stInitSubModulesException.etDiag											:= GD.ET_Diag.UnexpectedProgramBehavior;
stInitSubModulesException.udiDiagExt										:= ET_DiagExt.InitSubModulesException;
stInitSubModulesException.sDiagExt											:= FC_EtDiagExtToString(stInitSubModulesException.udiDiagExt);
stInitSubModulesException.sMsg												:= '';	(* Replaced on usage *)
stInitSubModulesException.udiModuleId										:= iq_stStandardModuleItf.i_udiModuleId;
stInitSubModulesException.sModuleName										:= iq_stStandardModuleItf.i_sModuleName;
stInitSubModulesException.stReaction.axReaction[TPL.ET_Reaction.AsyncStop]	:= TRUE;
stInitSubModulesException.etSource											:= TPL.ET_ExceptionSource.NodeModule;
stInitSubModulesException.timDelayTime										:= T#0MS;
stInitSubModulesException.wHmiAttributes									:= 0;
stInitSubModulesException.xAutoQuit											:= FALSE;

stIsDriveVirtualException.etDiag											:= GD.ET_Diag.InputParameterInvalid;
stIsDriveVirtualException.udiDiagExt										:= ET_DiagExt.ifMulticarrierSegmentsInvalid ;
stIsDriveVirtualException.sDiagExt											:= FC_EtDiagExtToString(stIsDriveVirtualException.udiDiagExt);
stIsDriveVirtualException.sMsg												:= '';	(* Replaced on usage *)
stIsDriveVirtualException.udiModuleId										:= iq_stStandardModuleItf.i_udiModuleId;
stIsDriveVirtualException.sModuleName										:= iq_stStandardModuleItf.i_sModuleName;
stIsDriveVirtualException.stReaction.axReaction[TPL.ET_Reaction.AsyncStop]	:= TRUE;
stIsDriveVirtualException.etSource											:= TPL.ET_ExceptionSource.NodeModule;
stIsDriveVirtualException.timDelayTime										:= T#0MS;
stIsDriveVirtualException.wHmiAttributes									:= 0;
stIsDriveVirtualException.xAutoQuit											:= FALSE;

(*------------------------------------------------------------------------------------------*)
(* Init User Exceptions *)

	// TPL.ET_Reaction.AsyncStop
	// TPL.ET_Reaction.SyncStopEL
	// TPL.ET_Reaction.SyncStopEH
	// TPL.ET_Reaction.StopEndOfCycle
	// TPL.ET_Reaction.MainsContactorOff

(*------------------------------------------------------------------------------------------*)
stUserException1.etDiag													:= GD.ET_Diag.ExecutionAborted;
stUserException1.udiDiagExt												:= ET_DiagExtUser.Exception1FromEquipmentModule;
stUserException1.sDiagExt												:= FC_EtDiagExtUserToString(stUserException1.udiDiagExt);
stUserException1.sMsg													:= 'User Exception 1';
stUserException1.udiModuleId											:= iq_stStandardModuleItf.i_udiModuleId;
stUserException1.sModuleName											:= iq_stStandardModuleItf.i_sModuleName;
stUserException1.stReaction.axReaction[TPL.Gc_udiUserReactionOffset+2]	:= TRUE;
stUserException1.etSource												:= TPL.ET_ExceptionSource.User;
stUserException1.timDelayTime											:= T#0MS;
stUserException1.wHmiAttributes											:= 0;
stUserException1.xAutoQuit												:= FALSE;

stUserException2.etDiag													:= GD.ET_Diag.ExecutionAborted;
stUserException2.udiDiagExt												:= ET_DiagExtUser.Exception2FromEquipmentModule;
stUserException2.sDiagExt												:= FC_EtDiagExtUserToString(stUserException2.udiDiagExt);
stUserException2.sMsg													:= 'User Exception 2';
stUserException2.udiModuleId											:= iq_stStandardModuleItf.i_udiModuleId;
stUserException2.sModuleName											:= iq_stStandardModuleItf.i_sModuleName;
stUserException2.stReaction.axReaction[TPL.Gc_udiUserReactionOffset+2]	:= TRUE;
stUserException2.etSource												:= TPL.ET_ExceptionSource.User;
stUserException2.timDelayTime											:= T#0MS;
stUserException2.wHmiAttributes											:= 0;
stUserException2.xAutoQuit												:= FALSE;

(* End of system generated code, could be modified for your application *)
END_ACTION

ACTION Init_Reactions:
(* System generated code, only to be changed by experienced programmers *)
IF c_udiNumberOfSubModules < 1 THEN
	RETURN;
END_IF

(* Change of default reactions only on demand *)
(* Compare SR MainMachine Action Init_Reactions *)

xInitReactionsException := FALSE;

(*****************************************************************************************************************************************************)
(* Init ReactionTranslationMode *)

TPL.FC_InitReactionTranslationMode(	i_udiNumberOfSubModules			:= c_udiNumberOfSubModules,
									i_petReactionTranslationMode	:= ADR(aetReactionTranslationMode),
									q_etDiag						=> etDiag,
									q_etDiagExt						=> etDiagExtTPL);
							
IF etDiag <> GD.ET_Diag.Ok AND NOT xInitReactionsException THEN
	xInitReactionsException := TRUE;
	
	stInitReactionsException.sMsg := PDL.FC_MultiConcat(i_sString1 := 'InitReactionTranslationMode - ', 
														i_sString2 := GD.FC_EtDiagToString(i_etDiag := etDiag), 
														i_sString3 := ' - ', 
														i_sString4 := TPL.FC_EtDiagExtToString(i_etDiagExt := etDiagExtTPL));
END_IF	

(*****************************************************************************************************************************************************)
(* Init ReactionTranslationTable *)	

TPL.FC_InitReactionTranslationTable(i_udiNumberOfSubModules			:= c_udiNumberOfSubModules,
									i_pstReactionTranslationTable	:= ADR(aastReactionTranslationTable),
									q_etDiag						=> etDiag,
									q_etDiagExt						=> etDiagExtTPL);
									
IF etDiag <> GD.ET_Diag.Ok AND NOT xInitReactionsException THEN
	xInitReactionsException := TRUE;
	
	stInitReactionsException.sMsg := PDL.FC_MultiConcat(i_sString1 := 'InitReactionTranslationTable - ', 
														i_sString2 := GD.FC_EtDiagToString(i_etDiag := etDiag), 
														i_sString3 := ' - ', 
														i_sString4 := TPL.FC_EtDiagExtToString(i_etDiagExt := etDiagExtTPL));
END_IF		

(*****************************************************************************************************************************************************)
(* Init ReactionTranslationJobs *)	
					
TPL.FC_InitReactionTranslationJobs( i_udiNumberOfSubModules			:= c_udiNumberOfSubModules,
									i_pstReactionTranslationJobs	:= ADR(astReactionTranslationJobs),
									q_etDiag						=> etDiag,
									q_etDiagExt						=> etDiagExtTPL);
						
IF etDiag <> GD.ET_Diag.Ok AND NOT xInitReactionsException THEN
	xInitReactionsException := TRUE;
	
	stInitReactionsException.sMsg := PDL.FC_MultiConcat(i_sString1 := 'InitReactionTranslationJobs - ', 
														i_sString2 := GD.FC_EtDiagToString(i_etDiag := etDiag), 
														i_sString3 := ' - ', 
														i_sString4 := TPL.FC_EtDiagExtToString(i_etDiagExt := etDiagExtTPL));
END_IF		

(*****************************************************************************************************************************************************)
(* Set exception if any exception occurred *)
fbExceptionHandler.SetException(i_xExceptionActive	:= xInitReactionsException, 
								iq_stException		:= stInitReactionsException, 
								iq_stExceptionList	:= iq_stExceptionList);
		
xInitSuccessful := xInitSuccessful AND NOT xInitReactionsException;

etDiag := GD.ET_Diag.Ok;
(* End of system generated code, only to be changed by experienced programmers *)
END_ACTION

ACTION ModuleFaults:
(* System generated code, could be modified for your application *)
(* User Exception *)
fbExceptionHandler.SetException(	i_xExceptionActive	:= xModuleUserException1,
									iq_stException		:= stUserException1,
									iq_stExceptionList	:= iq_stExceptionList,
									q_etDiag			=> ,
									q_etDiagExt			=> ,
									q_sMsg				=> );

fbExceptionHandler.SetException(	i_xExceptionActive	:= xModuleUserException2,
									iq_stException		:= stUserException2,
									iq_stExceptionList	:= iq_stExceptionList,
									q_etDiag			=> ,
									q_etDiagExt			=> ,
									q_sMsg				=> );

(* end of System generated code, could be modified for your application *)
END_ACTION

METHOD RegisterLoggerPoint
VAR_INPUT
	i_ifParent	: APL.IF_LoggerPoint;
	i_sName		: STRING[80];
END_VAR
VAR_OUTPUT
	q_etDiag	: GD.ET_Diag := GD.ET_Diag.Ok;
	q_etDiagExt	: ET_DiagExt := ET_DiagExt.Ok;
END_VAR
fbLoggerPoint.RegisterLoggerPoint(	i_ifParent	:= i_ifParent,
									i_sName		:= i_sName,
									i_sType		:= 'Node Module',
									i_sSource	:= 'Program',
									q_etDiag	=> ,
									q_etDiagExt	=> );
END_METHOD

ACTION InitModule_Action:
(* This step is used for initialisations after being enabled *)

(* System generated code, could be modified for your application *)
Init_Exceptions();
(* End of system generated code, could be modified for your application *)

(* System generated code, do not change without consulting 'Schneider Electric Automation GmbH' - otherwise you risk instability!!!*)
xInitSuccessful := TRUE;
xIsDriveVirtualException := FALSE;

iq_stStandardModuleItf.q_xActive		:= TRUE;
iq_stStandardModuleItf.q_xReady			:= FALSE;
iq_stStandardModuleItf.q_etDiag			:= GD.ET_Diag.Ok;
iq_stStandardModuleItf.q_udiDiagExt		:= ET_DiagExt.Initializing;
iq_stStandardModuleItf.q_sDiagExt		:= FC_EtDiagExtToString(ET_DiagExt.Initializing);
iq_stStandardModuleItf.q_sMsg			:= '';
			
Init_SubModules();
Init_CmdTables();
Init_Reactions();
UpdateStructs();
(* End of system generated code, do not change without consulting 'Schneider Electric Automation GmbH' - otherwise you risk instability!!!*)

(* System generated code, could be modified for your application *)
fbModuleController.RegisterLoggerPoint(	i_ifParent	:= fbLoggerPoint,
										i_sName		:= 'ModuleController',
										q_etDiag	=> ,
										q_etDiagExt	=> );
fbExceptionHandler.RegisterLoggerPoint(	i_ifParent	:= fbLoggerPoint,
										i_sName		:= 'ExceptionHandler',
										q_etDiag	=> ,
										q_etDiagExt	=> );
										
Init_Master();
(* End of system generated code, could be modified for your application *)

(* Application specific code *)
(* ToDo: Add your application specific code here *)
;
(* End of application specific code *)
END_ACTION

ACTION Input_Action:
(* System generated code, do not change without consulting 'Schneider Electric Automation GmbH' - otherwise you risk instability!!!*)
UpdateStructs();
(* End of system generated code, do not change without consulting 'Schneider Electric Automation GmbH' - otherwise you risk instability!!!*)
END_ACTION

ACTION Logger_Action:
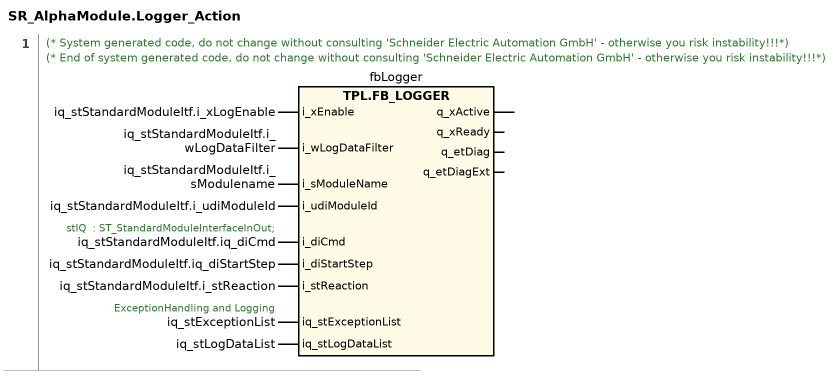
// NETWORK 1
// 					(* System generated code, do not change without consulting 'Schneider Electric Automation GmbH' - otherwise you risk instability!!!*)
// (* End of system generated code, do not change without consulting 'Schneider Electric Automation GmbH' - otherwise you risk instability!!!*)
//
//   fbLogger: Logging related variables
//   iq_stStandardModuleItf.iq_diCmd: stIQ : ST_StandardModuleInterfaceInOut;
//   iq_stExceptionList: ExceptionHandling and Logging
fbLogger(
    i_xEnable := iq_stStandardModuleItf.i_xLogEnable,
    i_wLogDataFilter := iq_stStandardModuleItf.i_wLogDataFilter,
    i_sModuleName := iq_stStandardModuleItf.i_sModulename,
    i_udiModuleId := iq_stStandardModuleItf.i_udiModuleId,
    i_diCmd := iq_stStandardModuleItf.iq_diCmd,
    i_diStartStep := iq_stStandardModuleItf.iq_diStartStep,
    i_stReaction := iq_stStandardModuleItf.i_stReaction,
    iq_stExceptionList := iq_stExceptionList,
    iq_stLogDataList := iq_stLogDataList); // TPL.FB_LOGGER
END_ACTION

ACTION Logic_active:
Check_RTB();
END_ACTION

ACTION Output_Active:
(* System generated code, only to be changed by experienced programmers *)
IF iq_stStandardModuleItf.q_udiSubModuleInException <> 0 THEN
	iq_stStandardModuleItf.q_etDiag		:= GD.ET_Diag.Ok;
	iq_stStandardModuleItf.q_udiDiagExt	:= ET_DiagExt.SubModuleInException;
	iq_stStandardModuleItf.q_sDiagExt		:= FC_EtDiagExtToString(ET_DiagExt.SubModuleInException);
	iq_stStandardModuleItf.q_sMsg			:= '';
ELSE
	IF etDiagModuleController = GD.ET_Diag.Ok THEN
		iq_stStandardModuleItf.q_etDiag	:= etDiagModuleController;
		iq_stStandardModuleItf.q_sMsg		:= sMsgModuleController;
		
		CASE etDiagExtModuleController OF
			TPL.ET_DiagExt.DeactivatingSubModules : 
				iq_stStandardModuleItf.q_udiDiagExt	:= ET_DiagExt.DeactivatingSubModules;
				iq_stStandardModuleItf.q_sDiagExt		:= FC_EtDiagExtToString(ET_DiagExt.DeactivatingSubModules);
			TPL.ET_DiagExt.Disabled : 
				iq_stStandardModuleItf.q_udiDiagExt	:= ET_DiagExt.Disabled;
				iq_stStandardModuleItf.q_sDiagExt		:= FC_EtDiagExtToString(ET_DiagExt.Disabled);
			TPL.ET_DiagExt.ExecuteStep : 
				iq_stStandardModuleItf.q_udiDiagExt	:= ET_DiagExt.ExecuteStep;
				iq_stStandardModuleItf.q_sDiagExt		:= FC_EtDiagExtToString(ET_DiagExt.ExecuteStep);
			TPL.ET_DiagExt.Initializing : 
				iq_stStandardModuleItf.q_udiDiagExt	:= ET_DiagExt.Initializing;
				iq_stStandardModuleItf.q_sDiagExt		:= FC_EtDiagExtToString(ET_DiagExt.Initializing);
			TPL.ET_DiagExt.WaitAtNegativeStep : 
				iq_stStandardModuleItf.q_udiDiagExt	:= ET_DiagExt.WaitAtNegativeStep;
				iq_stStandardModuleItf.q_sDiagExt		:= FC_EtDiagExtToString(ET_DiagExt.WaitAtNegativeStep);
			TPL.ET_DiagExt.WaitCmdsDone : 
				iq_stStandardModuleItf.q_udiDiagExt	:= ET_DiagExt.WaitCmdsDone;
				iq_stStandardModuleItf.q_sDiagExt		:= FC_EtDiagExtToString(ET_DiagExt.WaitCmdsDone);
			TPL.ET_DiagExt.WaitForCmd : 
				iq_stStandardModuleItf.q_udiDiagExt	:= ET_DiagExt.WaitForCmd;
				iq_stStandardModuleItf.q_sDiagExt		:= FC_EtDiagExtToString(ET_DiagExt.WaitForCmd);
			ELSE
				iq_stStandardModuleItf.q_etDiag		:= GD. ET_Diag.UnexpectedProgramBehavior;
				iq_stStandardModuleItf.q_udiDiagExt	:= ET_DiagExt.UnknownStateModuleController;
				iq_stStandardModuleItf.q_sDiagExt		:= FC_EtDiagExtToString(ET_DiagExt.UnknownStateModuleController);
		END_CASE
	ELSE
		iq_stStandardModuleItf.q_etDiag		:= GD.ET_Diag.DiagActive;
		iq_stStandardModuleItf.q_udiDiagExt	:= ET_DiagExt.ModuleControllerException;
		iq_stStandardModuleItf.q_sDiagExt		:= FC_EtDiagExtToString(ET_DiagExt.ModuleControllerException);
		iq_stStandardModuleItf.q_sMsg			:= PDL.FC_MultiConcat(	i_sString1 := GD.FC_EtDiagToString(i_etDiag := etDiagModuleController), 
																			i_sString2 := ' - ',
																			i_sString3 := TPL.FC_EtDiagExtToString(etDiagExtModuleController), 
																			i_sString4 := '');
	END_IF
END_IF

(* End of system generated code, only to be changed by experienced programmers *)
END_ACTION

ACTION Start_Action:
(* This step is active until the machine is being enabled *)

(* System generated code, do not change without consulting 'Schneider Electric Automation GmbH' - otherwise you risk instability!!! *)
iq_stStandardModuleItf.q_xActive			:= FALSE;
iq_stStandardModuleItf.q_xReady				:= FALSE;

iq_stStandardModuleItf.q_etDiag				:= GD.ET_Diag.Ok;
iq_stStandardModuleItf.q_udiDiagExt			:= ET_DiagExt.Disabled;
iq_stStandardModuleItf.q_sDiagExt			:= FC_EtDiagExtToString(iq_stStandardModuleItf.q_udiDiagExt);
iq_stStandardModuleItf.q_sMsg				:= '';

iq_stStandardModuleItf.q_dwModuleType		:= TPL.ET_ModuleType.NodeModule;
iq_stStandardModuleItf.q_sModuleTypeName	:= 'NodeModule';
iq_stStandardModuleItf.q_udiModuleVersion	:= 1;	
(* End of system generated code, do not change without consulting 'Schneider Electric Automation GmbH' - otherwise you risk instability!!! *)

(* System generated code, to be changed by experienced programmers *)
IF iq_stStandardModuleItf.iq_diCmd <> 0 AND NOT iq_stStandardModuleItf.i_xEnable THEN
	iq_stStandardModuleItf.iq_diCmd := 0;
END_IF
(* End of system generated code, to be changed by experienced programmers *)

(* Application specific code *)
(* ToDo: Add your application specific code here *)
;
(* End of application specific code *)
END_ACTION

ACTION SubModules_Action:
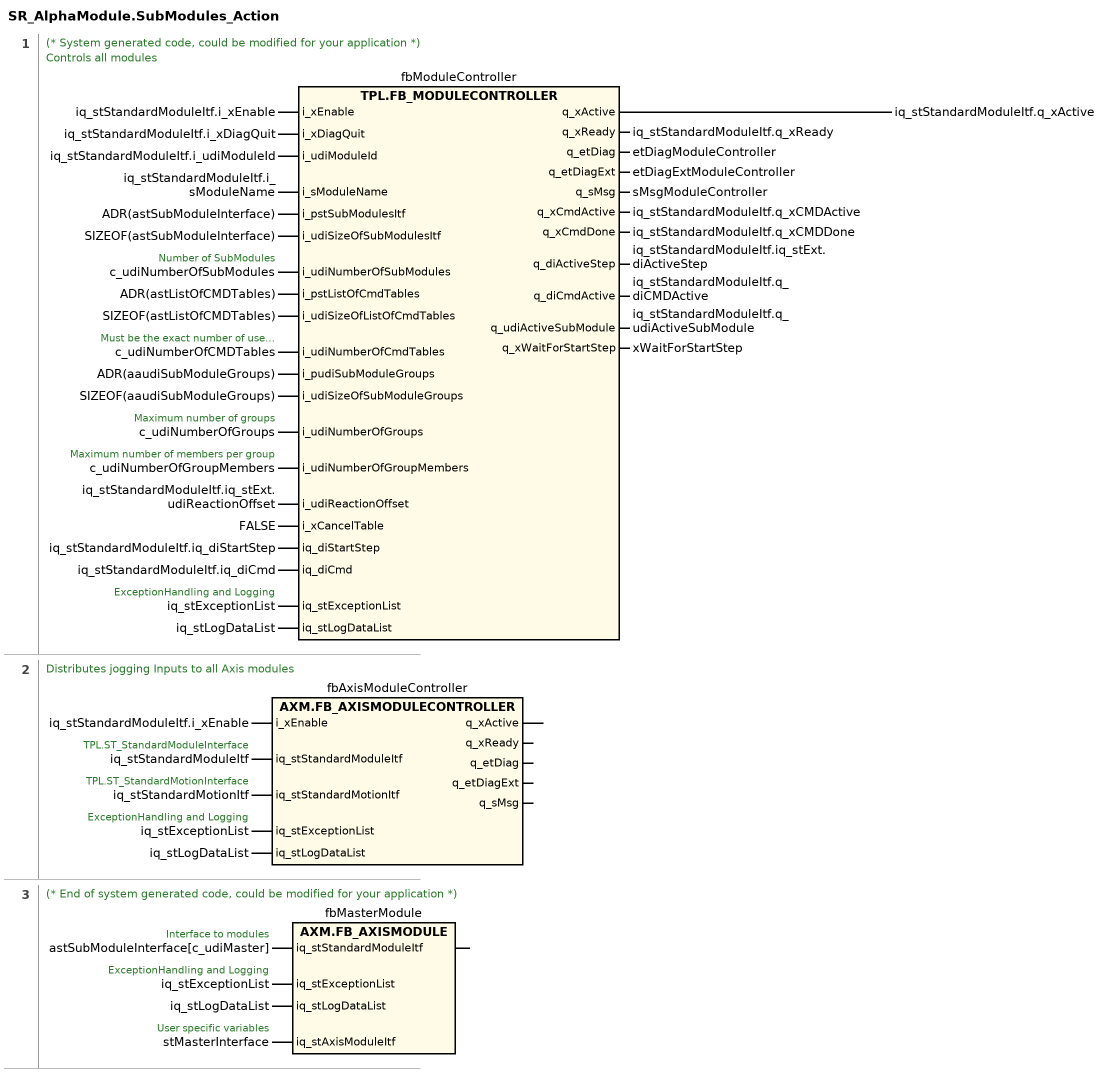
// NETWORK 1
// 					(* System generated code, could be modified for your application *)
// Controls all modules
//
//   fbModuleController: Modules related variables
//   c_udiNumberOfSubModules: Number of SubModules
//   c_udiNumberOfCMDTables: Must be the exact number of used CmdTables!
//   c_udiNumberOfGroups: Maximum number of groups
//   c_udiNumberOfGroupMembers: Maximum number of members per group
//   iq_stExceptionList: ExceptionHandling and Logging
fbModuleController(
    i_xEnable := iq_stStandardModuleItf.i_xEnable,
    i_xDiagQuit := iq_stStandardModuleItf.i_xDiagQuit,
    i_udiModuleId := iq_stStandardModuleItf.i_udiModuleId,
    i_sModuleName := iq_stStandardModuleItf.i_sModuleName,
    i_pstSubModulesItf := ADR(astSubModuleInterface),
    i_udiSizeOfSubModulesItf := SIZEOF(astSubModuleInterface),
    i_udiNumberOfSubModules := c_udiNumberOfSubModules,
    i_pstListOfCmdTables := ADR(astListOfCMDTables),
    i_udiSizeOfListOfCmdTables := SIZEOF(astListOfCMDTables),
    i_udiNumberOfCmdTables := c_udiNumberOfCMDTables,
    i_pudiSubModuleGroups := ADR(aaudiSubModuleGroups),
    i_udiSizeOfSubModuleGroups := SIZEOF(aaudiSubModuleGroups),
    i_udiNumberOfGroups := c_udiNumberOfGroups,
    i_udiNumberOfGroupMembers := c_udiNumberOfGroupMembers,
    i_udiReactionOffset := iq_stStandardModuleItf.iq_stExt.udiReactionOffset,
    i_xCancelTable := FALSE,
    iq_diStartStep := iq_stStandardModuleItf.iq_diStartStep,
    iq_diCmd := iq_stStandardModuleItf.iq_diCmd,
    iq_stExceptionList := iq_stExceptionList,
    iq_stLogDataList := iq_stLogDataList,
    q_xReady => iq_stStandardModuleItf.q_xReady,
    q_etDiag => etDiagModuleController,
    q_etDiagExt => etDiagExtModuleController,
    q_sMsg => sMsgModuleController,
    q_xCmdActive => iq_stStandardModuleItf.q_xCMDActive,
    q_xCmdDone => iq_stStandardModuleItf.q_xCMDDone,
    q_diActiveStep => iq_stStandardModuleItf.iq_stExt.diActiveStep,
    q_diCmdActive => iq_stStandardModuleItf.q_diCMDActive,
    q_udiActiveSubModule => iq_stStandardModuleItf.q_udiActiveSubModule,
    q_xWaitForStartStep => xWaitForStartStep); // TPL.FB_MODULECONTROLLER
iq_stStandardModuleItf.q_xActive := fbModuleController.q_xActive;

// NETWORK 2
// Distributes jogging Inputs to all Axis modules
//   iq_stStandardModuleItf: TPL.ST_StandardModuleInterface
//   iq_stStandardMotionItf: TPL.ST_StandardMotionInterface
//   iq_stExceptionList: ExceptionHandling and Logging
fbAxisModuleController(
    i_xEnable := iq_stStandardModuleItf.i_xEnable,
    iq_stStandardModuleItf := iq_stStandardModuleItf,
    iq_stStandardMotionItf := iq_stStandardMotionItf,
    iq_stExceptionList := iq_stExceptionList,
    iq_stLogDataList := iq_stLogDataList); // AXM.FB_AXISMODULECONTROLLER

// NETWORK 3
// (* End of system generated code, could be modified for your application *)
//   astSubModuleInterface[c_udiMaster]: Interface to modules
//   iq_stExceptionList: ExceptionHandling and Logging
//   stMasterInterface: User specific variables
fbMasterModule(
    iq_stStandardModuleItf := astSubModuleInterface[c_udiMaster],
    iq_stExceptionList := iq_stExceptionList,
    iq_stLogDataList := iq_stLogDataList,
    iq_stAxisModuleItf := stMasterInterface); // AXM.FB_AXISMODULE
END_ACTION

ACTION UpdateStructs:
(* System generated code, do not change without consulting 'Schneider Electric Automation GmbH' - otherwise you risk instability!!! *)
fbDetectOnlineChange(	i_xEnable	:= TRUE, 
						i_xDetect	:= TRUE, 
						q_xActive	=> xDetectOnlineChangeActive, 
						q_xReady	=> xDetectOnlineChangeReady, 
						q_etDiag	=> etDetectOnlineChangeDiag, 
						q_etDiagExt	=> etDetectOnlineChangeDiagExt, 
						q_sMsg		=> sDetectOnlineChangeMsg, 
						q_xChange	=> );
						
IF(NOT fbDetectOnlineChange.q_xChange) THEN
	RETURN;
END_IF

iq_stStandardModuleItf.iq_stExt.udiNumberOfSubModules 		:= c_udiNumberOfSubModules;
iq_stStandardModuleItf.iq_stExt.dwSubModulesItf		 		:= ADR(astSubModuleInterface);
iq_stStandardModuleItf.iq_stExt.pdwSubModulesAddItf		 	:= ADR(adwSubModuleAddInterfaces);
iq_stStandardModuleItf.iq_stExt.pstListOfCmdTables			:= ADR(astListOfCmdTables);
iq_stStandardModuleItf.iq_stExt.udiNumberOfCmdTables		:= c_udiNumberOfCmdTables;
(* End of system generated code, do not change without consulting 'Schneider Electric Automation GmbH' - otherwise you risk instability!!! *)

(* System generated code, could be modified for your application *)
xUpdateStructsException := FALSE;

//-------------------------------------------------------------------------------------------------------------------
//-- Update CmdTable - Prepare 
	//
	TPL.FC_UpdateCmdTableListElement(	i_pstListofCmdTables	:= ADR(astListOfCmdTables),
										i_udiNumberOfCmdTables	:= c_udiNumberOfCmdTables,
										i_diCmd					:= ET_Cmd.Prepare,
										i_pstCmdTable			:= ADR(astPrepareTable),
										q_etDiag				=> etDiag,
										q_etDiagExt				=> etDiagExtTPL);
										
	IF etDiag <> GD.ET_Diag.Ok AND NOT xUpdateStructsException THEN
		xUpdateStructsException := TRUE;
		
		stUpdateStructsException.sMsg := PDL.FC_MultiConcat(i_sString1 := 'Update CmdTable: Prepare - ', 
															i_sString2 := GD.FC_EtDiagToString(i_etDiag := etDiag), 
															i_sString3 := ' - ', 
															i_sString4 := TPL.FC_EtDiagExtToString(i_etDiagExt := etDiagExtTPL));
	END_IF										

//-------------------------------------------------------------------------------------------------------------------
//-- Update CmdTable - Auto 
	//
	TPL.FC_UpdateCmdTableListElement(	i_pstListofCmdTables	:= ADR(astListOfCmdTables),
										i_udiNumberOfCmdTables	:= c_udiNumberOfCmdTables,
										i_diCmd					:= ET_Cmd.Auto,
										i_pstCmdTable			:= ADR(astAutoTable),
										q_etDiag				=> etDiag,
										q_etDiagExt				=> etDiagExtTPL);
										
	IF etDiag <> GD.ET_Diag.Ok AND NOT xUpdateStructsException THEN
		xUpdateStructsException := TRUE;
		
		stUpdateStructsException.sMsg := PDL.FC_MultiConcat(i_sString1 := 'Update CmdTable: Auto - ', 
															i_sString2 := GD.FC_EtDiagToString(i_etDiag := etDiag), 
															i_sString3 := ' - ', 
															i_sString4 := TPL.FC_EtDiagExtToString(i_etDiagExt := etDiagExtTPL));
	END_IF		

//-------------------------------------------------------------------------------------------------------------------
//-- Update CmdTable - Manual 
	//
	TPL.FC_UpdateCmdTableListElement(	i_pstListofCMDTables	:= ADR(astListofCMDTables),
										i_udiNumberOfCMDTables	:= c_udiNumberOfCMDTables,
										i_diCMD					:= ET_Cmd.Manual,
										i_pstCMDTable			:= ADR(astManualTable),
										q_etDiag				=> etDiag,
										q_etDiagExt				=> etDiagExtTPL);
										
	IF etDiag <> GD.ET_Diag.Ok AND NOT xUpdateStructsException THEN
		xUpdateStructsException := TRUE;
		
		stUpdateStructsException.sMsg := PDL.FC_MultiConcat(i_sString1 := 'Update CmdTable: Manual - ', 
															i_sString2 := GD.FC_EtDiagToString(i_etDiag := etDiag), 
															i_sString3 := ' - ', 
															i_sString4 := TPL.FC_EtDiagExtToString(i_etDiagExt := etDiagExtTPL));
	END_IF		

//-------------------------------------------------------------------------------------------------------------------
//-- Update CmdTable - Stop 
	//
	TPL.FC_UpdateCmdTableListElement(	i_pstListofCMDTables	:= ADR(astListofCMDTables),
										i_udiNumberOfCMDTables	:= c_udiNumberOfCMDTables,
										i_diCMD					:= ET_Cmd.Stop,
										i_pstCMDTable			:= ADR(astStopTable),
										q_etDiag				=> etDiag,
										q_etDiagExt				=> etDiagExtTPL);
										
	IF etDiag <> GD.ET_Diag.Ok AND NOT xUpdateStructsException THEN
		xUpdateStructsException := TRUE;
		
		stUpdateStructsException.sMsg := PDL.FC_MultiConcat(i_sString1 := 'Update CmdTable: Stop - ', 
															i_sString2 := GD.FC_EtDiagToString(i_etDiag := etDiag), 
															i_sString3 := ' - ', 
															i_sString4 := TPL.FC_EtDiagExtToString(i_etDiagExt := etDiagExtTPL));
	END_IF		

//-------------------------------------------------------------------------------------------------------------------
//-- Update CmdTable - Start 
	//
	TPL.FC_UpdateCmdTableListElement(	i_pstListofCMDTables	:= ADR(astListofCMDTables),
										i_udiNumberOfCmdTables	:= c_udiNumberOfCMDTables,
										i_diCMD					:= ET_Cmd.Start,
										i_pstCMDTable			:= ADR(astStartTable),
										q_etDiag				=> etDiag,
										q_etDiagExt				=> etDiagExtTPL);
										
	IF etDiag <> GD.ET_Diag.Ok AND NOT xUpdateStructsException THEN
		xUpdateStructsException := TRUE;
		
		stUpdateStructsException.sMsg := PDL.FC_MultiConcat(i_sString1 := 'Update CmdTable: Start - ', 
															i_sString2 := GD.FC_EtDiagToString(i_etDiag := etDiag), 
															i_sString3 := ' - ', 
															i_sString4 := TPL.FC_EtDiagExtToString(i_etDiagExt := etDiagExtTPL));
	END_IF		

//-------------------------------------------------------------------------------------------------------------------
//-- Update CmdTable - Abort 
	//
	TPL.FC_UpdateCmdTableListElement(	i_pstListofCMDTables	:= ADR(astListofCMDTables),
										i_udiNumberOfCmdTables	:= c_udiNumberOfCmdTables,
										i_diCMD					:= ET_Cmd.Abort,
										i_pstCMDTable			:= ADR(astAbortTable),
										q_etDiag				=> etDiag,
										q_etDiagExt				=> etDiagExtTPL);
										
	IF etDiag <> GD.ET_Diag.Ok AND NOT xUpdateStructsException THEN
		xUpdateStructsException := TRUE;
		
		stUpdateStructsException.sMsg := PDL.FC_MultiConcat(i_sString1 := 'Update CmdTable: Abort - ', 
															i_sString2 := GD.FC_EtDiagToString(i_etDiag := etDiag), 
															i_sString3 := ' - ', 
															i_sString4 := TPL.FC_EtDiagExtToString(i_etDiagExt := etDiagExtTPL));
	END_IF		

//-------------------------------------------------------------------------------------------------------------------
//-- Update CmdTable - Hold 
	//
	TPL.FC_UpdateCmdTableListElement(	i_pstListofCMDTables	:= ADR(astListofCMDTables),
										i_udiNumberOfCmdTables	:= c_udiNumberOfCmdTables,
										i_diCMD					:= ET_Cmd.Hold,
										i_pstCMDTable			:= ADR(astHoldTable),
										q_etDiag				=> etDiag,
										q_etDiagExt				=> etDiagExtTPL);
										
	IF etDiag <> GD.ET_Diag.Ok AND NOT xUpdateStructsException THEN
		xUpdateStructsException := TRUE;
		
		stUpdateStructsException.sMsg := PDL.FC_MultiConcat(i_sString1 := 'Update CmdTable: Hold - ', 
															i_sString2 := GD.FC_EtDiagToString(i_etDiag := etDiag), 
															i_sString3 := ' - ', 
															i_sString4 := TPL.FC_EtDiagExtToString(i_etDiagExt := etDiagExtTPL));
	END_IF		

//-------------------------------------------------------------------------------------------------------------------
//-- Update CmdTable - BrakeRelease 
	//
	TPL.FC_UpdateCmdTableListElement(	i_pstListofCMDTables	:= ADR(astListofCMDTables),
										i_udiNumberOfCMDTables	:= c_udiNumberOfCMDTables,
										i_diCMD					:= ET_Cmd.BrakeRelease,
										i_pstCMDTable			:= ADR(astBrakeReleaseTable),
										q_etDiag				=> etDiag,
										q_etDiagExt				=> etDiagExtTPL);
										
	IF etDiag <> GD.ET_Diag.Ok AND NOT xUpdateStructsException THEN
		xUpdateStructsException := TRUE;
		
		stUpdateStructsException.sMsg := PDL.FC_MultiConcat(i_sString1 := 'Update CmdTable: BrakeRelease - ', 
															i_sString2 := GD.FC_EtDiagToString(i_etDiag := etDiag), 
															i_sString3 := ' - ', 
															i_sString4 := TPL.FC_EtDiagExtToString(i_etDiagExt := etDiagExtTPL));
	END_IF		
									
//-------------------------------------------------------------------------------------------------------------------
//-- Update AddInterface - Master 
	//

	AXM.FC_UpdateAddInterfaceStruct(	i_pdwSubModuleAddInterfaces	:= ADR(adwSubModuleAddInterfaces),
										i_udiSubModuleConstant		:= c_udiMaster,
										iq_stAxisModuleItf			:= stMasterInterface,
										q_etDiag					=> etDiag,
										q_etDiagExt					=> etDiagExtAXM);
										
	IF etDiag <> GD.ET_Diag.Ok AND NOT xUpdateStructsException THEN
		xUpdateStructsException := TRUE;
		
		stUpdateStructsException.sMsg := PDL.FC_MultiConcat(i_sString1 := 'Update AddInterface: Master - ', 
															i_sString2 := GD.FC_EtDiagToString(i_etDiag := etDiag), 
															i_sString3 := ' - ', 
															i_sString4 := AXM.FC_EtDiagExtToString(i_etDiagExt := etDiagExtAXM));
	END_IF		

//-------------------------------------------------------------------------------------------------------------------
//-- Update ILS Data 
	//
	// stMasterInterface.stEndless.pstIlsData	:= ADR(G_stIlsData);
	// stMasterInterface.stMultiCam.pstIlsData	:= ADR(G_stIlsData);

//-------------------------------------------------------------------------------------------------------------------
//-- Set exception if any exception occurred *)

fbExceptionHandler.SetException(i_xExceptionActive	:= xUpdateStructsException, 
								iq_stException		:= stUpdateStructsException, 
								iq_stExceptionList	:= iq_stExceptionList);
					
xInitSuccessful := xInitSuccessful AND NOT xUpdateStructsException;

etDiag := GD.ET_Diag.Ok;
(* End of system generated code, could be modified for your application *)
END_ACTION

END_PROGRAM

// LMC_PacDrive/Application/TemplateFullProgrammingFramework/Tools/FC_IsDriveVirtual
FUNCTION FC_IsDriveVirtual : BOOL
VAR_INPUT
	i_ifDrive	: SystemConfigurationItf.IF_Drive;
END_VAR

VAR_OUTPUT
	q_etDiag	: GD.ET_Diag := GD.ET_Diag.Ok;
	q_etDiagExt	: ET_DiagExt := ET_DiagExt.Ok;
	q_sMsg		: STRING[80];
END_VAR

VAR
	xSuccess						: BOOL;
	ifSercosDeviceIdentification	: SystemConfigurationItf.IF_SercosDeviceIdentification; 
END_VAR

IF i_ifDrive = 0 THEN
	q_etDiag	:= GD.ET_Diag.InputParameterInvalid;
	q_etDiagExt	:= ET_DiagExt.ifMulticarrierSegmentsInvalid ;
	q_sMsg		:= 'FC_IsDriveVirtual: i_ifDrive not set';		
ELSE
	xSuccess := __QUERYINTERFACE(i_ifDrive, ifSercosDeviceIdentification);
	IF NOT xSuccess OR ifSercosDeviceIdentification = 0 THEN
		q_etDiag	:= GD.ET_Diag.InputParameterInvalid;
		q_etDiagExt	:= ET_DiagExt.ifMulticarrierSegmentsInvalid ;
		q_sMsg		:= Standard.CONCAT(i_ifDrive.Name, ' - IF_SercosDeviceIdentification not implemented');						
	ELSE
		IF ifSercosDeviceIdentification.WorkingState = 0 THEN	// Drive is virtual
			FC_IsDriveVirtual := TRUE;
		ELSE
			FC_IsDriveVirtual := FALSE;
		END_IF
	END_IF
END_IF

END_FUNCTION

// LMC_PacDrive/Application/TemplateFullProgrammingFramework/Tools/FC_SetDeadTimeCompensation
FUNCTION FC_SetDeadTimeCompensation : BOOL
VAR_INPUT
	i_stSubModuleInterfaceMain		: AXM.ST_Main;
END_VAR
VAR
(* Init related variables *)	
	stLogicalAddressMaster			: SystemConfigurationItf.ST_LogicalAddress;
	lrShaftRefDelay					: LREAL;
	lrPositionDelay					: LREAL; 
	diResult						: DINT;	

END_VAR

IF i_stSubModuleInterfaceMain.i_ifMaster <> 0 AND i_stSubModuleInterfaceMain.i_ifDrive <> 0 THEN	
	stLogicalAddressMaster := i_stSubModuleInterfaceMain.i_ifMaster.stLogicalAddress;
	IF (stLogicalAddressMaster.udiType = SYSTEMINTERFACE.P_ENC_TYPE.udiType) OR			(* Physical encoder *)
		(stLogicalAddressMaster.udiType = SYSTEMINTERFACE.INC_IN_TYPE.udiType) OR		(* Incremental	encoder *)
		(stLogicalAddressMaster.udiType = SYSTEMINTERFACE.SYN_DIN_TYPE.udiType) OR		(* SyncMaster encoder *)
		(stLogicalAddressMaster.udiType = SYSTEMINTERFACE.C2C_ENC_IN_TYPE.udiType) OR	(* C2C Encoder input *)
		(stLogicalAddressMaster.udiType = SYSTEMINTERFACE.V_ENC_TYPE.udiType) THEN		(* Virtual master encoder *)
		
		stLogicalAddressMaster := i_stSubModuleInterfaceMain.i_ifDrive.stLogicalAddress;
		stLogicalAddressMaster.udiParameterId := 16#00A2;
		diResult := SYSTEMINTERFACE.FC_GetParameter(i_stLogAdr	:= stLogicalAddressMaster,
													i_dwBuffer	:= ADR(lrShaftRefDelay),
													i_diSize	:= SIZEOF(lrShaftRefDelay));
		IF diResult = 0 THEN
			i_stSubModuleInterfaceMain.iq_lencEncoder.Delay := -lrShaftRefDelay;
		END_IF
	ELSIF (stLogicalAddressMaster.udiType = SYSTEMINTERFACE.INC_IN3_TYPE.udiType) THEN  (* IncIn via TM5 TM5SE1IC20005 *)
		stLogicalAddressMaster := i_stSubModuleInterfaceMain.i_ifDrive.stLogicalAddress;
		stLogicalAddressMaster.udiParameterId := 16#00A2;
		diResult := SYSTEMINTERFACE.FC_GetParameter(i_stLogAdr	:= stLogicalAddressMaster,
													i_dwBuffer	:= ADR(lrShaftRefDelay),
													i_diSize	:= SIZEOF(lrShaftRefDelay));
		IF diResult = 0 THEN
			i_stSubModuleInterfaceMain.iq_lencEncoder.Delay := -lrShaftRefDelay;
			stLogicalAddressMaster := i_stSubModuleInterfaceMain.i_ifMaster.stLogicalAddress;
			stLogicalAddressMaster.udiParameterId := 16#008E; 					(* Parameter PositionDelay of TM5SE1IC20005 *)
			diResult := SYSTEMINTERFACE.FC_GetParameter(i_stLogAdr	:= stLogicalAddressMaster,
														i_dwBuffer	:= ADR(lrPositionDelay),
														i_diSize	:= SIZEOF(lrPositionDelay));		
			IF diResult = 0 THEN
				i_stSubModuleInterfaceMain.iq_lencEncoder.Delay := -(lrShaftRefDelay + (-lrPositionDelay)) ;
			END_IF
		END_IF
	END_IF
END_IF

IF diResult = 0 THEN
	FC_SetDeadTimeCompensation := TRUE;
END_IF

END_FUNCTION

// LMC_PacDrive/Application/TemplateFullProgrammingFramework/ProjectDiagnostics/FC_EtDiagExtUserToString
FUNCTION FC_EtDiagExtUserToString : STRING[80]
VAR_INPUT
	i_etDiagExt : ET_DiagExtUser;
END_VAR
VAR_OUTPUT
	q_etDiag	: GD.ET_Diag := GD.ET_Diag.Ok;
	q_etDiagExt	: ET_DiagExt := ET_DiagExt.Ok;
END_VAR
VAR
END_VAR

CASE i_etDiagExt OF
	ET_DiagExtUser.Exception1FromEquipmentModule	: FC_EtDiagExtUserToString := 'Exception1FromEquipmentModule';
	ET_DiagExtUser.Exception2FromEquipmentModule	: FC_EtDiagExtUserToString := 'Exception2FromEquipmentModule';
	
	ET_DiagExtUser.Exception1FromMain				: FC_EtDiagExtUserToString := 'Exception1FromMain';
	ET_DiagExtUser.Exception2FromMain				: FC_EtDiagExtUserToString := 'Exception2FromMain';
	ET_DiagExtUser.Exception3FromMain				: FC_EtDiagExtUserToString := 'Exception3FromMain';
	ET_DiagExtUser.Exception4FromMain				: FC_EtDiagExtUserToString := 'Exception4FromMain';
	ET_DiagExtUser.Exception5FromMain				: FC_EtDiagExtUserToString := 'Exception5FromMain';
ELSE
	FC_EtDiagExtUserToString := CONCAT('Unkown ET_DiagExtUser ', UDINT_TO_STRING(i_etDiagExt));
		
	q_etDiag	:= GD.ET_Diag.InputParameterInvalid;
	q_etDiagExt	:= ET_DiagExt.UnknownDiagExtUser;
END_CASE

END_FUNCTION

// LMC_PacDrive/Application/TemplateFullProgrammingFramework/EquipmentModules/SR_BravoModule
PROGRAM SR_BravoModule

VAR CONSTANT
(* Standard related constants *)
	c_udiNumberOfGroups				: UDINT := 3;			(* Maximum number of groups *)
	c_udiNumberOfGroupMembers		: UDINT := 10;			(* Maximum number of members per group *)

	c_udiNumberOfCmdTables			: UDINT := 8;			(* Must be the exact number of used CMDTables! *)
	c_udiNumberOfCmdSteps			: UDINT := 16;			(* Make sure that the number of commands/ Steps  that each table
																   contains does not exceed the c_diNumberOfCMDSteps variable.*)

(* Definition group of modules *)
	c_udiBravoGroup1				: UDINT := 2001;		(* Name of module group  1 *)
	c_udiBravoGroup2				: UDINT := 2002;		(* Name of module group  2 *)

(* System generated code, could be modified for your application *)
	c_udiNumberOfSubModules			: UDINT := 2;			(* Number of axis modules *)
	c_udiSlave1						: UDINT := 1;
	c_udiSlave2						: UDINT := 2;
(* End of system generated code, could be modified for your application *)
END_VAR

VAR (* User specific variables *)
	stSlave1Interface				: AXM.ST_ModuleInterface;
	fbSlave1Module					: AXM.FB_AxisModule;
	
	stSlave2Interface				: AXM.ST_ModuleInterface;
	fbSlave2Module					: AXM.FB_AxisModule;
	
	fbAxisModuleController			: AXM.FB_AxisModuleController;
END_VAR

VAR_INPUT
(* Master of BravoModule *)
	i_ifMaster						: SystemConfigurationItf.IF_Master;
END_VAR

VAR_IN_OUT
(* TPL.ST_StandardModuleInterface *)	
	iq_stStandardModuleItf			: TPL.ST_StandardModuleInterface;
	
(* TPL.ST_StandardMotionInterface *)		
	iq_stStandardMotionItf			: TPL.ST_StandardMotionInterface;
	
(* ExceptionHandling and Logging *)	
	iq_stExceptionList				: TPL.ST_ExceptionList;
	iq_stLogDataList				: TPL.ST_LogDataList;
END_VAR

VAR
	xInitSuccessful : BOOL := TRUE;
		
(* Standard related variables *)
	astSubModuleInterface			: ARRAY[1..c_udiNumberOfSubModules] OF TPL.ST_StandardModuleInterface;		(* Interface to modules *)
	aaudiSubModuleGroups			: ARRAY[1..c_udiNumberOfGroups,1..c_udiNumberOfGroupMembers] OF UDINT;
	adwSubModuleAddInterfaces		: ARRAY[1..c_udiNumberOfSubModules] OF DWORD;
(* Modules related variables *)
	fbModuleController				: TPL.FB_ModuleController;
	etDiagModuleController			: GD.ET_Diag;
	etDiagExtModuleController		: TPL.ET_DiagExt;
	sMsgModuleController			: STRING[80];
	xWaitForStartStep				: BOOL;
	
	astListOfCmdTables				: ARRAY [1..c_udiNumberOfCmdTables] OF TPL.ST_CmdTable;
	udiTableIndex					: UDINT;
	udiStepIndex					: UDINT;
	diStep							: DINT;

	astPrepareTable					: ARRAY [1..c_udiNumberOfCmdSteps] OF TPL.ST_Cmd;		(* Relating  Cmd table *)
	astAutoTable					: ARRAY [1..c_udiNumberOfCmdSteps] OF TPL.ST_Cmd;		(* Relating  Cmd table *)
	astManualTable					: ARRAY [1..c_udiNumberOfCmdSteps] OF TPL.ST_Cmd;		(* Relating  Cmd table *)
	astHoldTable					: ARRAY [1..c_udiNumberOfCmdSteps] OF TPL.ST_Cmd;		(* Relating  Cmd table *)
	astStartTable					: ARRAY [1..c_udiNumberOfCmdSteps] OF TPL.ST_Cmd;		(* Relating  Cmd table *)
	astStopTable					: ARRAY [1..c_udiNumberOfCmdSteps] OF TPL.ST_Cmd;		(* Relating  Cmd table *)
	astBrakeReleaseTable			: ARRAY [1..c_udiNumberOfCmdSteps] OF TPL.ST_Cmd;		(* Relating  Cmd table *)
	astAbortTable					: ARRAY [1..c_udiNumberOfCmdSteps] OF TPL.ST_Cmd;		(* Relating  Cmd table *)

(* ExceptionHandling related variables *)
	fbExceptionHandler				: TPL.FB_ExceptionHandler2;

	aetReactionTranslationMode		: ARRAY[1..c_udiNumberOfSubModules] OF TPL.ET_ReactionTranslationMode;
	aastReactionTranslationTable	: ARRAY[1..c_udiNumberOfSubModules,1..TPL.Gc_udiMaxNumberOfReactions] OF TPL.ST_Reaction;
	astReactionTranslationJobs		: ARRAY[1..c_udiNumberOfSubModules] OF TPL.ST_ReactionTranslationJobs;
	
(* Exception declaration *)
	stUserException1				: TPL.ST_Exception;
	stUserException2				: TPL.ST_Exception;
	xModuleUserException1			: BOOL;
	xModuleUserException2			: BOOL;
	
	stUpdateStructsException		: TPL.ST_Exception;
	xUpdateStructsException			: BOOL;
	
	stInitReactionsException		: TPL.ST_Exception;
	xInitReactionsException			: BOOL;
	
	stInitSubModulesException		: TPL.ST_Exception;
	xInitSubModulesException		: BOOL;
	
	stIsDriveVirtualException		: TPL.ST_Exception;
	xIsDriveVirtualException		: BOOL;

(* Logging related variables *)
	fbLogger						: TPL.FB_Logger;
	fbLoggerPoint					: APL.FB_LoggerPoint;

(* OnlineChange related variables *)
	fbDetectOnlineChange			: TPL.FB_DetectOnlineChange;
	xDetectOnlineChangeActive		: BOOL; 
	xDetectOnlineChangeReady		: BOOL; 
	etDetectOnlineChangeDiag		: GD.ET_Diag;
	etDetectOnlineChangeDiagExt		: TPL.ET_DiagExt; 
	sDetectOnlineChangeMsg			: STRING[80];
	
(* Init related variables *)	
	stLogicalAddressMaster			: SystemConfigurationItf.ST_LogicalAddress;
	lrShaftRefDelay					: LREAL;
	diResult						: DINT;	
	
	xDriveIsVirtual					: BOOL;	
	
(* POU-Feedback related variables *)	
	etDiag			: GD.ET_Diag;
	etDiagExt		: ET_DiagExt;
	etDiagExtTPL	: TPL.ET_DiagExt;
	etDiagExtAXM	: AXM.ET_DiagExt;
	sMsgBuffer		: STRING[80];
	xReInit			: BOOL; 	
	
(* Check RTB  *)
	diStateRTB						: DINT := 0;
	xRTBFailureFlag					: BOOL;
	udiCount						: UDINT;
	xModulesActive					: BOOL;
	xModulesNotActive				: BOOL;	
	
END_VAR

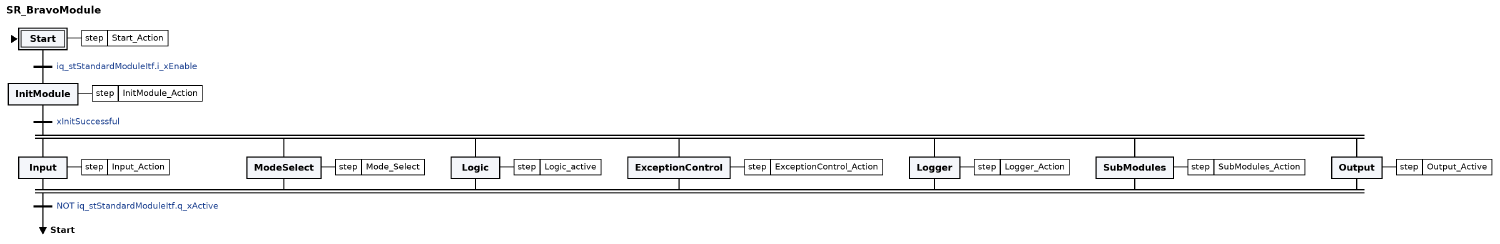
INITIAL_STEP Start:
    Start_Action(N);  // step action
END_STEP
TRANSITION FROM Start TO InitModule
    := iq_stStandardModuleItf.i_xEnable;
END_TRANSITION
STEP InitModule:
    InitModule_Action(N);  // step action
END_STEP
TRANSITION FROM InitModule TO (Input, ModeSelect, Logic, ExceptionControl, Logger, SubModules, Output)
    := xInitSuccessful;
END_TRANSITION
STEP Input:
    Input_Action(N);  // step action
END_STEP
STEP ModeSelect:
    Mode_Select(N);  // step action
END_STEP
STEP Logic:
    Logic_active(N);  // step action
END_STEP
STEP ExceptionControl:
    ExceptionControl_Action(N);  // step action
END_STEP
STEP Logger:
    Logger_Action(N);  // step action
END_STEP
STEP SubModules:
    SubModules_Action(N);  // step action
END_STEP
STEP Output:
    Output_Active(N);  // step action
END_STEP
TRANSITION FROM (Input, ModeSelect, Logic, ExceptionControl, Logger, SubModules, Output) TO Start
    := NOT iq_stStandardModuleItf.q_xActive;
END_TRANSITION

ACTION Check_RTB:
(*
check RTB State
If RTB failure, all axis modules will be disabled.
After restart RTB, then all axis modules will be enabled again and the axes positions will be restored.
after home ok, opmode could be selected 
*)
(*########################################################################################*)

(* check RTB failure *)
IF Sercos_Master.State <> 4
AND NOT xRTBFailureFlag THEN

	xRTBFailureFlag := TRUE;
	
		(* disable axes modules *)
		FOR udiCount := 1 TO c_udiNumberOfSubModules DO
			
			(* axis module detection *)
			IF astSubModuleInterface[udiCount].q_dwModuleType = TPL.ET_ModuleType.AxisModule THEN
				astSubModuleInterface[udiCount].i_xEnable 		:= FALSE;	(* disable axes modules *)
			END_IF
		END_FOR
		
		diStateRTB := 10;

ELSIF Sercos_Master.State = 4 THEN	(* RTB ok *)
	xRTBFailureFlag := FALSE;
END_IF

(************************************************************************************************************************)
	CASE diStateRTB OF

	0:;	(* wait *)

	10:	(* wait for restart RTB *)

		IF Sercos_Master.State > 0
		AND Sercos_Master.State  <> 4 THEN
			xReInit								 := TRUE;		(* set marker reinit active *)
			diStateRTB := 20;
		END_IF

	20:	(* wait for RTB ready and ErrorQuit. / wait till AxesModules are disabled / --> restart axes modules *)
		FOR udiCount := 1 TO c_udiNumberOfSubModules DO
			
			(* axis module detection *)
			IF astSubModuleInterface[udiCount].q_dwModuleType = TPL.ET_ModuleType.AxisModule THEN
				IF astSubModuleInterface[udiCount].q_xActive THEN	(* module active *)
					xModulesNotActive 							:= FALSE;
					EXIT;
				ELSIF NOT astSubModuleInterface[udiCount].q_xActive THEN	(* module not active *)
					xModulesNotActive 							:= TRUE;
				END_IF
			END_IF
		END_FOR

		IF Sercos_Master.State = 4
		AND xModulesNotActive
		AND iq_stStandardModuleItf.i_xDiagQuit THEN
		
			FOR udiCount := 1 TO c_udiNumberOfSubModules DO
				(* axis module detection *)
				IF astSubModuleInterface[udiCount].q_dwModuleType = TPL.ET_ModuleType.AxisModule THEN
					astSubModuleInterface[udiCount].i_xEnable	 := TRUE;	(* enable axes modules *)
				END_IF
			END_FOR
			diStateRTB := 30;
		END_IF

	30:	(* wait for axes modules active *)

		FOR udiCount := 1 TO c_udiNumberOfSubModules DO
			
			(* axis module detection *)
			IF astSubModuleInterface[udiCount].q_dwModuleType = TPL.ET_ModuleType.AxisModule THEN
				IF NOT astSubModuleInterface[udiCount].q_xActive THEN	(* module not active *)
					xModulesActive 								:= FALSE;
					EXIT;
				ELSIF astSubModuleInterface[udiCount].q_xActive THEN	(* module active *)
					xModulesActive 								:= TRUE;
				END_IF
			END_IF
		END_FOR

		IF xModulesActive THEN	(* all axis modules active *)
			diStateRTB := 40;
		END_IF

	40:	(* Reinit ready  *)

		xReInit									:= FALSE;		(* reset marker reinit active *)
		diStateRTB := 0;

	END_CASE
END_ACTION

ACTION Init_Slave1:
//--- System generated code, could be modified for your application ---------------------------------------------------------

//--- Standard interface ---------------------------------------------------------
	//
	astSubModuleInterface[c_udiSlave1].i_sModuleName		:= CONCAT(STR1 := iq_stStandardModuleItf.i_sModuleName, STR2 := ': Slave1');
	
	astSubModuleInterface[c_udiSlave1].i_xLogEnable			:= 	TRUE;
	astSubModuleInterface[c_udiSlave1].i_wLogDataFilter		:= 	UDINT_TO_WORD(TPL.ET_LogDataFilter.ModuleDefault);
	
	fbSlave1Module.RegisterLoggerPoint(	i_ifParent	:= fbLoggerPoint,
										i_sName		:= 'Slave1',
										q_etDiag	:= ,
										q_etDiagExt	:= );
//
//--- Master, Drive& LEnc ---------------------------------------------------------
	//
	stSlave1Interface.stMain.i_ifMaster			:= i_ifMaster; 		//--- Master ----
	stSlave1Interface.stMain.i_ifDrive			:= DRV_Slave1;
	stSlave1Interface.stMain.iq_lencEncoder		:= LE_Slave1;
//
//--- Check if Drive is virtual ---------------------------------------------------------
	//
	xDriveIsVirtual := FC_IsDriveVirtual(	i_ifDrive	:= stSlave1Interface.stMain.i_ifDrive,
											q_etDiag	=> etDiag,
											q_etDiagExt	=> etDiagExt,
											q_sMsg		=> sMsgBuffer);

	IF etDiag <> GD.ET_Diag.Ok AND NOT xIsDriveVirtualException THEN
		stIsDriveVirtualException.etDiag 	:= etDiag;
		stIsDriveVirtualException.udiDiagExt:= etDiagExt;
		stIsDriveVirtualException.sDiagExt 	:= FC_EtDiagExtToString(etDiagExt);															
		stIsDriveVirtualException.sMsg 		:= sMsgBuffer;
		xIsDriveVirtualException 			:= TRUE;
	END_IF
	
	fbExceptionHandler.SetException(i_xExceptionActive	:= xIsDriveVirtualException, 
									iq_stException		:= stIsDriveVirtualException, 
									iq_stExceptionList	:= iq_stExceptionList);
					
	xInitSuccessful := xInitSuccessful AND NOT xIsDriveVirtualException;
	etDiag := GD.ET_Diag.Ok;
//
//--- Set DeadTime compensation parameters depending on used type of Master ---------------------------------------------------------
	FC_SetDeadTimeCompensation(i_stSubModuleInterfaceMain := stSlave1Interface.stMain);
	
//
//--- Set Velocity Parameters ---------------------------------------------------------
	stSlave1Interface.stMain.i_lrMotionActiveVelLimit						:= 15.0;	//--- Limit for max. velocity of astAxisModuleInterface to switch output AxisMove in Units/s ---------------------------------------------------------
	stSlave1Interface.stMain.i_etMotionActiveVelType						:= AXM.ET_MotionActiveVelType.Velocity;
	
	stSlave1Interface.stMain.stReducedVelocity.i_xEnableReducedVelocity		:= FALSE;
	stSlave1Interface.stMain.stReducedVelocity.i_xOnlyLimitCheck			:= FALSE;
	stSlave1Interface.stMain.stReducedVelocity.i_lrMaxReducedVelocity		:= 50.0;

	
	
//
//--- Stop Parameters ---------------------------------------------------------
	stSlave1Interface.stMain.i_timMasterStop								:= T#1S;
	stSlave1Interface.stMain.i_xHwLimitPos									:= FALSE;
	stSlave1Interface.stMain.i_xHwLimitNeg									:= FALSE;
	stSlave1Interface.stMain.i_xStart										:= FALSE;


//
//--- Set Homing Mode ---------------------------------------------------------
	//
	IF xDriveIsVirtual THEN
		stSlave1Interface.stHome.i_etMode := PDL.ET_HomeMode.SetPosAxisAndLogEncoderPosition;			//--- Homing Mode  in case of virtual axis ---------------------------------------------------------
	ELSE
		stSlave1Interface.stHome.i_etMode := PDL.ET_HomeMode.PosDirectionPosEdgeTp;						//--- Homing Mode in case of real axis ---------------------------------------------------------
	END_IF
		
	
	stSlave1Interface.stHome.i_xEnableInitAbsReadPos := FALSE;		(* TRUE : Restores the AxisPosition depending on the stHome.etMode
																			  If stHome.i_etMode is equal to PDL.ET_HomeMode.RestorePosFromAxisEncoder or 
																			  to PDL.ET_HomeMode.WriteAxisEncoder, the encoder of the axis is read,
																			  or else the position will be restored from the retain area *)
																			  
	stSlave1Interface.stHome.stSetpos.iq_pstRestorePosRetain := ADR(Grp_stRestorePositionAxis2);
	
	stSlave1Interface.stHome.i_xResetHomeOk := FALSE;
//
//--- Homing mode Sensor:
	(*	PDL.ET_HomeMode.PosDirectionPosEdgeSensor
		PDL.ET_HomeMode.NegDirectionPosEdgeSensor
		PDL.ET_HomeMode.NegDirectionNegEdgeSensor
		PDL.ET_HomeMode.PosDirectionNegEdgeSensor	*)

	stSlave1Interface.stHome.stSensor.i_lrHomePosition			:= 0.0;			//--- Position at the end of homing in units ---------------------------------------------------------
	stSlave1Interface.stHome.stSensor.i_lrVel					:= 10.0;		//--- Homing ceiling velocity in units/s ---------------------------------------------------------
	stSlave1Interface.stHome.stSensor.i_lrAcc					:= 1000.0;		//--- Homing acceleration in units/s^2 ---------------------------------------------------------
	stSlave1Interface.stHome.stSensor.i_lrDec					:= 1000.0;		//--- Homing deceleration in units/s^2 ---------------------------------------------------------
	stSlave1Interface.stHome.stSensor.i_lrJerk					:= 10000.0;		//--- Homing jerk in units/s^3 ---------------------------------------------------------
	stSlave1Interface.stHome.stSensor.i_lrOffset				:= 0.0;			//--- Offset from home signal in units ---------------------------------------------------------
	stSlave1Interface.stHome.stSensor.i_lrMaxTravel				:= 720.0;		//--- Max. travel for referencing by normal input ---------------------------------------------------------
	stSlave1Interface.stHome.stSensor.i_xRotativeSystem			:= FALSE;		//--- Rotative system true or false for referencing by normal input ---------------------------------------------------------
	stSlave1Interface.stHome.stSensor.i_xSensor					:= FALSE;		//--- Input for home signal. Can be a signal from a controller input. Has to be written cyclic. ---------------------------------------------------------

//--- Homing mode LimitSwitch:
	(*	PDL.ET_HomeMode.PosDirectionPosEdgeHWLimitPos		normally open contact / Closing contact
		PDL.ET_HomeMode.NegDirectionPosEdgeHWLimitNeg		normally open contact / Closing contact
		PDL.ET_HomeMode.NegDirectionNegEdgeHWLimitNeg		normally closed contact / Opening contact  
		PDL.ET_HomeMode.PosDirectionNegEdgeHWLimitPos		normally closed contact / Opening contact *)

	stSlave1Interface.stHome.stLimitSwitch.i_lrHomePosition		:= 0.0;			//--- Position at the end of homing in units ---------------------------------------------------------
	stSlave1Interface.stHome.stLimitSwitch.i_lrVel				:= 10.0;		//--- Homing ceiling velocity in units/s ---------------------------------------------------------
	stSlave1Interface.stHome.stLimitSwitch.i_lrLowVel			:= 5.0;			//--- Homing low ceiling velocity in units/s ---------------------------------------------------------
	stSlave1Interface.stHome.stLimitSwitch.i_lrAcc				:= 1000.0;		//--- Homing acceleration in units/s^2 ---------------------------------------------------------
	stSlave1Interface.stHome.stLimitSwitch.i_lrDec				:= 1000.0;		//--- Homing deceleration in units/s^2 ---------------------------------------------------------
	stSlave1Interface.stHome.stLimitSwitch.i_lrJerk				:= 10000.0;		//--- Homing jerk in units/s^3 ---------------------------------------------------------
	stSlave1Interface.stHome.stLimitSwitch.i_lrOffset			:= 0.0;			//--- Offset from home signal in units ---------------------------------------------------------
	stSlave1Interface.stHome.stLimitSwitch.i_lrMaxTravel		:= 9999.0;		//--- Max. travel for referencing normal input as a hardware limit ---------------------------------------------------------

//--- Homing mode MoveOnPos:
	(*PDL.ET_HomeMode.MoveOnPosAbs *)

	stSlave1Interface.stHome.stMoveOnPos.i_lrTarget				:= 0.0;			//--- Position at the end of homing in units ---------------------------------------------------------
	stSlave1Interface.stHome.stMoveOnPos.i_lrVel				:= 10.0;		//--- Homing ceiling velocity in units/s ---------------------------------------------------------
	stSlave1Interface.stHome.stMoveOnPos.i_lrAcc				:= 1000.0;		//--- Homing acceleration in units/s^2 ---------------------------------------------------------
	stSlave1Interface.stHome.stMoveOnPos.i_lrDec				:= 1000.0;		//--- Homing deceleration in units/s^2 ---------------------------------------------------------
	stSlave1Interface.stHome.stMoveOnPos.i_lrJerk				:= 10000.0;		//--- Homing jerk in units/s^3 ---------------------------------------------------------
	stSlave1Interface.stHome.stMoveOnPos.i_lrPeriod				:= 0.0;			//--- Period of the axis ---------------------------------------------------------
	stSlave1Interface.stHome.stMoveOnPos.i_xRotativeSystem		:= FALSE;		//--- Rotative system true or false ---------------------------------------------------------

//--- Homing mode SetPos:
	(*	PDL.ET_HomeMode.SetPosAxisPosition 
		PDL.ET_HomeMode.SetPosLogEncoderPosition 
		PDL.ET_HomeMode.SetPosAxisAndLogEncoderPosition
		PDL.ET_HomeMode.RestorePosFromAxisEncoder 
		PDL.ET_HomeMode.RestorePosFromRetain 				*)

	stSlave1Interface.stHome.stSetpos.i_lrHomePosition			:= 0.0;			//--- Position at the end of homing in units ---------------------------------------------------------
	stSlave1Interface.stHome.stSetpos.i_lrEncoderPosition		:= 0.0;			//--- Encoder position in units after homing ---------------------------------------------------------
	stSlave1Interface.stHome.stSetpos.i_lrAbsEncOffset			:= 100.0;		//--- Distance to the jump of axis encoder in units  ---------------------------------------------------------
	stSlave1Interface.stHome.stSetpos.i_lrRestoreWindow			:= 180;			//--- How far can the drive be away from is correct position ---------------------------------------------------------
	stSlave1Interface.stHome.stSetpos.i_lrUserPeriod			:= 360;			//--- Period of the axis ---------------------------------------------------------

//--- Homing mode Torque:
	(*	PDL.ET_HomeMode.PosDirectionMaxTorque 
		PDL.ET_HomeMode.NegDirectionMaxTorque *)

	stSlave1Interface.stHome.stTorque.i_lrHomePosition			:= 0.0;			//--- Position at the end of homing in units ---------------------------------------------------------
	stSlave1Interface.stHome.stTorque.i_lrVel					:= 10.0;		//--- Homing ceiling velocity in units/s ---------------------------------------------------------
	stSlave1Interface.stHome.stTorque.i_lrAcc					:= 1000.0;		//--- Homing acceleration in units/s^2 ---------------------------------------------------------
	stSlave1Interface.stHome.stTorque.i_lrDec					:= 1000.0;		//--- Homing deceleration in units/s^2 ---------------------------------------------------------
	stSlave1Interface.stHome.stTorque.i_lrJerk					:= 10000.0;		//--- Homing jerk in units/s^3 ---------------------------------------------------------
	stSlave1Interface.stHome.stTorque.i_lrOffset				:= 0.0;			//--- Offset from home signal in units ---------------------------------------------------------
	stSlave1Interface.stHome.stTorque.i_lrMaxTravel				:= 9999.0;		//--- Max. travel for referencing by torque ---------------------------------------------------------
	stSlave1Interface.stHome.stTorque.i_lrMaxTorque				:= 0.0;			//--- Torque for stop in Nm / referencing by torque ---------------------------------------------------------
	stSlave1Interface.stHome.stTorque.i_diTorqueTime			:= 5;			//--- Time in msec to hold torque ---------------------------------------------------------

//--- Homing mode TouchProbe:
	(*	PDL.ET_HomeMode.PosDirectionPosEdgeTp 
		PDL.ET_HomeMode.NegDirectionPosEdgeTp 
		PDL.ET_HomeMode.NegDirectionNegEdgeTp 
		PDL.ET_HomeMode.PosDirectionNegEdgeTp *)

	stSlave1Interface.stHome.stTouchProbe.i_lrHomePosition		:= 0.0;			//--- Position at the end of homing in units ---------------------------------------------------------
	stSlave1Interface.stHome.stTouchProbe.i_lrVel				:= 100.0;		//--- Homing ceiling velocity in units/s ---------------------------------------------------------
	stSlave1Interface.stHome.stTouchProbe.i_lrAcc				:= 1000.0;		//--- Homing acceleration in units/s^2 ---------------------------------------------------------
	stSlave1Interface.stHome.stTouchProbe.i_lrDec				:= 1000.0;		//--- Homing deceleration in units/s^2 ---------------------------------------------------------
	stSlave1Interface.stHome.stTouchProbe.i_lrJerk				:= 10000.0;		//--- Homing jerk in units/s^3 ---------------------------------------------------------
	stSlave1Interface.stHome.stTouchProbe.i_lrOffset			:= 30.0;		//--- Offset from home signal in units ---------------------------------------------------------
	stSlave1Interface.stHome.stTouchProbe.i_lrMaxTravel			:= 720.0;		//--- Max. travel for referencing by TP ---------------------------------------------------------
	stSlave1Interface.stHome.stTouchProbe.i_xRotativeSystem		:= TRUE;		//--- Rotative system true or false for referencing by TP ---------------------------------------------------------
	stSlave1Interface.stHome.stTouchProbe.i_ifTouchProbe		:= TP_0;		//--- Input for TP ---------------------------------------------------------

//--- Homing mode WritePos:
	(*	PDL.ET_HomeMode.WriteAxisEncoder *)

	stSlave1Interface.stHome.stWritePos.i_lrHomePosition		:= 0.0;			//--- Position at the end of homing in units ---------------------------------------------------------
	stSlave1Interface.stHome.stWritePos.i_lrUserPeriod			:= 0.0;			//--- Calculates Drive.Position into period ( units ) ---------------------------------------------------------
	stSlave1Interface.stHome.stWritePos.i_lrAbsEncOffset		:= 100.0;		//--- Distance to the jump of axis encoder in units ---------------------------------------------------------

//
//--- Manual ---------------------------------------------------------
	//
	stSlave1Interface.stManual.i_lrVel								:= 50.0;			//--- Velocity in units/s ---------------------------------------------------------
	stSlave1Interface.stManual.i_lrAcc								:= 100.0;			//--- Acceleration in units/s^2 ---------------------------------------------------------
	stSlave1Interface.stManual.i_lrDec								:= 100.0;			//--- Deceleration in units/s^2 ---------------------------------------------------------
	stSlave1Interface.stManual.i_lrJerk								:= 1000.0;			//--- Jerk in units/s^3 ---------------------------------------------------------
	stSlave1Interface.stManual.i_lrMaxDistance						:= 120.0;			//--- Max pathlengths for one step in units ---------------------------------------------------------
	stSlave1Interface.stManual.i_xEndless							:= FALSE;			//--- TRUE: jogging endless; Position between the periode; FALSE: jogging in steps. Position can be out of periode ---------------------------------------------------------
	stSlave1Interface.stManual.i_lrPeriod							:= 360.0;			//--- Period of the axis ---------------------------------------------------------

//
//--- Cam ---------------------------------------------------------
	//
	stSlave1Interface.stMultiCam.i_etCSModeSlave					:= PDL.ET_MultiCamCsModeSlave.SetSlavePositionToFirstCamPosition;		//--- ColdStartMode Slave ---------------------------------------------------------
	stSlave1Interface.stMultiCam.i_etCSModeMaster					:= PDL.ET_MultiCamCsModeMaster.SetMasterPositionToFirstCamPosition;		//--- ColdStartMode Master ---------------------------------------------------------
	stSlave1Interface.stMultiCam.i_etWSMode							:= PDL.ET_MultiCamWsMode.StoredCamMoveAlwaysNoPositionCheck;			//--- WarmStartMode ---------------------------------------------------------
	stSlave1Interface.stMultiCam.i_lrWSWindow						:= 5.0;											//--- WarmStartWindow in Axis units ---------------------------------------------------------
	stSlave1Interface.stMultiCam.i_lrWSVel							:= 100.0;										//--- Velocity for WarmStart and CSModeSlave = PDL.ET_MultiCamCsModeSlave.MoveSlaveToFirstCamPosition in Units/s ---------------------------------------------------------
	stSlave1Interface.stMultiCam.i_lrWSAcc							:= 1000.0;										//--- Acceleration and deceleration for Warmstart and CSModeSlave = PDL.ET_MultiCamCsModeSlave.MoveSlaveToFirstCamPosition in Units/s^2 ---------------------------------------------------------
	stSlave1Interface.stMultiCam.i_lrWSJerk							:= 10000.0;										//--- Jerk for Warmstart and CSModeSlave = PDL.ET_MultiCamCsModeSlave.MoveSlaveToFirstCamPosition in units/s^3 ---------------------------------------------------------
	stSlave1Interface.stMultiCam.i_diTXend							:= 2*SYSTEMINTERFACE.FC_LzsTaskGetInterval();	//--- Time of XLowEnd and XHighEnd befor Xend or Xstart in msec---------------------------------------------------------
	stSlave1Interface.stMultiCam.i_lrInstantXLimMax					:= 0.0;											//--- Switch off position at 'InstantNewCam' ---------------------------------------------------------
	
	stSlave1Interface.stMultiCam.i_xEnableTabHandler				:= TRUE;										//--- TRUE: TabHandler is enabled ---------------------------------------------------------
	stSlave1Interface.stMultiCam.i_udiTableSelectNr					:= AXM.ET_ParId.User;							//--- Number of table which is used in the next cycle ---------------------------------------------------------
	
	stSlave1Interface.stMultiCam.i_xSetEncoderParameters			:= FALSE;										//--- TRUE: The parameters MasterId, FeedConstand, GearIn and GearOut will be copyed into LEnc object ---------------------------------------------------------
	stSlave1Interface.stMultiCam.i_xSetEncoderPosition				:= TRUE;										//--- TRUE: Manipulation of LEnc object on startup OpMode MultiCam ---------------------------------------------------------
	stSlave1Interface.stMultiCam.i_lrSetEncoderOffset				:= 0.0;											//--- Master encoder offset ---------------------------------------------------------
	stSlave1Interface.stMultiCam.i_xCheckEncoderPeriod				:= TRUE;										//--- TRUE: Check of encoder period = 0. If encoder period <> 0 -> Exception ---------------------------------------------------------
	
	//--- stSlave1Interface.stMultiCam.iq_xNewCam						:= FALSE;									//--- TRUE: A new DataStruct will be load for next cycle. Will be reset when new cycle is started in case of stMultiCam.i_xEnableTabHandler = FALSE. ---------------------------------------------------------
	//--- stSlave1Interface.stMultiCam.iq_xInstantNewCam				:= FALSE;									//--- TRUE: A new DataStruct will be load. It will be active at master position stMultiCam.i_lrInstantXLimMax. Will be reset when ne DataStruct is active ---------------------------------------------------------
	//--- stSlave1Interface.stMultiCam.iq_xChangeMaster				:= FALSE;										//--- TRUE: Switch to a new Master. Will be reset when done. ---------------------------------------------------------			
	
	//--- stSlave1Interface.stMultiCam.iq_stExt		;						//--- Extended In of the Multicam FB, can be used if needed! ---------------------------------------------------------
	
	//--- DataStruct used in CamDiagram_Slave1 ---------------------------------------------------------
	//stSlave1Interface.stMultiCam.iq_astMotionPar[AXM.ET_ParId.User].diNumberOfCamPoints		:= 4;	
	//stSlave1Interface.stMultiCam.iq_astMotionPar[AXM.ET_ParId.User].lrYPeriod				:= 0.0;
	//
	//stSlave1Interface.stMultiCam.iq_astMotionPar[AXM.ET_ParId.User].astCamPoint[0].lrX		:= 0.0;
	//stSlave1Interface.stMultiCam.iq_astMotionPar[AXM.ET_ParId.User].astCamPoint[0].lrY		:= 0.0;
	//stSlave1Interface.stMultiCam.iq_astMotionPar[AXM.ET_ParId.User].astCamPoint[0].lrM		:= 0.0;
	//stSlave1Interface.stMultiCam.iq_astMotionPar[AXM.ET_ParId.User].astCamPoint[0].etCamType	:= PDL.ET_CamType.Poly5Com;
	//stSlave1Interface.stMultiCam.iq_astMotionPar[AXM.ET_ParId.User].astCamPoint[1].lrX		:= 60.0;
	//stSlave1Interface.stMultiCam.iq_astMotionPar[AXM.ET_ParId.User].astCamPoint[1].lrY		:= 30.0;
	//stSlave1Interface.stMultiCam.iq_astMotionPar[AXM.ET_ParId.User].astCamPoint[1].lrM		:= 1.0;
	//stSlave1Interface.stMultiCam.iq_astMotionPar[AXM.ET_ParId.User].astCamPoint[1].etCamType	:= PDL.ET_CamType.Straight;
	//stSlave1Interface.stMultiCam.iq_astMotionPar[AXM.ET_ParId.User].astCamPoint[2].lrX		:= 240.0;
	//stSlave1Interface.stMultiCam.iq_astMotionPar[AXM.ET_ParId.User].astCamPoint[2].lrY		:= 210.0;
	//stSlave1Interface.stMultiCam.iq_astMotionPar[AXM.ET_ParId.User].astCamPoint[2].lrM		:= 1.0;
	//stSlave1Interface.stMultiCam.iq_astMotionPar[AXM.ET_ParId.User].astCamPoint[2].etCamType	:= PDL.ET_CamType.Poly5Com;
	//stSlave1Interface.stMultiCam.iq_astMotionPar[AXM.ET_ParId.User].astCamPoint[3].lrX		:= 360.0;
	//stSlave1Interface.stMultiCam.iq_astMotionPar[AXM.ET_ParId.User].astCamPoint[3].lrY		:= 0.0;
	//stSlave1Interface.stMultiCam.iq_astMotionPar[AXM.ET_ParId.User].astCamPoint[3].lrM		:= 0.0;
	//stSlave1Interface.stMultiCam.iq_astMotionPar[AXM.ET_ParId.User].astCamPoint[3].etCamType	:= PDL.ET_CamType.Poly5Com;
	
	stSlave1Interface.stMultiCam.iq_astMotionPar[AXM.ET_ParId.Idle].diUserTableId	:= UDINT_TO_DINT(AXM.ET_ParId.Idle);
	stSlave1Interface.stMultiCam.iq_astMotionPar[AXM.ET_ParId.Start].diUserTableId	:= UDINT_TO_DINT(AXM.ET_ParId.Start);
	stSlave1Interface.stMultiCam.iq_astMotionPar[AXM.ET_ParId.Cont].diUserTableId	:= UDINT_TO_DINT(AXM.ET_ParId.Cont);
	stSlave1Interface.stMultiCam.iq_astMotionPar[AXM.ET_ParId.Stop].diUserTableId	:= UDINT_TO_DINT(AXM.ET_ParId.Stop);
	stSlave1Interface.stMultiCam.iq_astMotionPar[AXM.ET_ParId.User].diUserTableId	:= UDINT_TO_DINT(AXM.ET_ParId.User);


	//--- ILS Data --------------------------------------------------------
	//---
	//stSlave1Interface.stMultiCam.i_udiIlsSlaveNumber													:= 1;
	//
	//G_stIlsData.i_stRunTime.astSlaveLimits[stSlave1Interface.stMultiCam.i_udiIlsSlaveNumber].lrPosVel	:= 1000.0;
	//G_stIlsData.i_stRunTime.astSlaveLimits[stSlave1Interface.stMultiCam.i_udiIlsSlaveNumber].lrNegVel	:= -1000.0;
	//G_stIlsData.i_stRunTime.astSlaveLimits[stSlave1Interface.stMultiCam.i_udiIlsSlaveNumber].lrPosAcc	:= 10000.0;
	//G_stIlsData.i_stRunTime.astSlaveLimits[stSlave1Interface.stMultiCam.i_udiIlsSlaveNumber].lrNegAcc	:= -10000.0;
	//
	//G_stIlsData.i_astCamData[stSlave1Interface.stMultiCam.i_udiIlsSlaveNumber].diNumberOfMasterPeriods	:= 1;	
	//G_stIlsData.i_astCamData[stSlave1Interface.stMultiCam.i_udiIlsSlaveNumber].diMasterPeriodInit		:= 1;
	//G_stIlsData.i_astCamData[stSlave1Interface.stMultiCam.i_udiIlsSlaveNumber].lrXOffset				:= 0.0;
	//
	//stSlave1Interface.stMultiCam.pstIlsData																:= ADR(G_stIlsData);
//
//--- Endless ---------------------------------------------------------
	//
	stSlave1Interface.stEndless.i_lrVel								:= 100.0;			//--- Velocity in Units/s ---------------------------------------------------------
	stSlave1Interface.stEndless.i_lrAcc								:= 1000.0;			//--- Acceleration in Units/s^2 ---------------------------------------------------------
	stSlave1Interface.stEndless.i_lrDec								:= 1000.0;			//--- Deceleration in Units/s^2 ---------------------------------------------------------
	stSlave1Interface.stEndless.i_lrJerk							:= 10000.0;			//--- Jerk in units/s^3 ---------------------------------------------------------
	stSlave1Interface.stEndless.i_lrPeriod							:= 360.0;			//--- Period one cycle in units ---------------------------------------------------------
	stSlave1Interface.stEndless.i_lrStopPosition					:= 0.5;				//--- Stop position in units ---------------------------------------------------------
//
//--- Endless ILS ---------------------------------------------------------
	//
	//G_stIlsData.i_stConfig.diNumberOfSlaves							:= 0;
	//G_stIlsData.i_stConfig.diPositionGridSize						:= 500;
	//G_stIlsData.i_stConfig.diTimeGridSize							:= 50;
	//G_stIlsData.i_stConfig.lrHysteresis								:= 20;
	//
	//G_stIlsData.i_stRunTime.iMasterAverageVelocityCycles			:= 10;
	//G_stIlsData.i_stRunTime.lrMasterMaxAbsVel						:= 100.0;
	//G_stIlsData.i_stRunTime.lrMasterMaxAbsAcc						:= 1000.0;
	//G_stIlsData.i_stRunTime.lrMasterMaxAbsJerk						:= 10000.0;
	//G_stIlsData.i_stRunTime.xActivateLimitation						:= TRUE;
	//
	//stSlave1Interface.stEndless.pstIlsData							:= ADR(G_stIlsData);
//
//--- Pos ---------------------------------------------------------
	//
	stSlave1Interface.stPos.i_etPosMode								:= SYSTEMINTERFACE.ET_PosMode.Relative;			//--- SYSTEMINTERFACE.ET_PosMode.Endless, SYSTEMINTERFACE.ET_PosMode.Relative, SYSTEMINTERFACE.ET_PosMode.Absolute ---------------------------------------------------------
	stSlave1Interface.stPos.i_lrTarget								:= -360.0;										//--- Target position or distance in Units ---------------------------------------------------------
	stSlave1Interface.stPos.i_lrVel									:= 100.0;										//--- Ceiling velocity in Units/s ---------------------------------------------------------
	stSlave1Interface.stPos.i_lrAcc									:= 3600.0;										//--- Acceleration in Units/s^2 ---------------------------------------------------------
	stSlave1Interface.stPos.i_lrDec									:= 3600.0;										//--- Deceleration in Units/s^2 ---------------------------------------------------------
	stSlave1Interface.stPos.i_lrJerk								:= 36000.0;										//--- Jerk in units/s^3 ---------------------------------------------------------

	//--- stSlave1Interface.stPos.i_xStop								:= FALSE;
//
//--- End of system generated code, could be modified for your application ---------------------------------------------------------
END_ACTION

ACTION Init_Slave2:
//--- System generated code, could be modified for your application ---------------------------------------------------------

//--- Standard interface ---------------------------------------------------------
	//
	astSubModuleInterface[c_udiSlave2].i_sModuleName		:= CONCAT(STR1 := iq_stStandardModuleItf.i_sModuleName, STR2 := ': Slave2');
	
	astSubModuleInterface[c_udiSlave2].i_xLogEnable			:= 	TRUE;
	astSubModuleInterface[c_udiSlave2].i_wLogDataFilter		:= 	UDINT_TO_WORD(TPL.ET_LogDataFilter.ModuleDefault);
	
	fbSlave2Module.RegisterLoggerPoint(	i_ifParent	:= fbLoggerPoint,
										i_sName		:= 'Slave2',
										q_etDiag	:= ,
										q_etDiagExt	:= );
//
//--- Master, Drive& LEnc ---------------------------------------------------------
	//
	stSlave2Interface.stMain.i_ifMaster			:= i_ifMaster; 		//--- Master ----
	stSlave2Interface.stMain.i_ifDrive			:= DRV_Slave2;
	stSlave2Interface.stMain.iq_lencEncoder		:= LE_Slave2;
	
	
//
//--- Check if Drive is virtual ---------------------------------------------------------
	//
	xDriveIsVirtual := FC_IsDriveVirtual(	i_ifDrive	:= stSlave2Interface.stMain.i_ifDrive,
											q_etDiag	=> etDiag,
											q_etDiagExt	=> etDiagExt,
											q_sMsg		=> sMsgBuffer);

	IF etDiag <> GD.ET_Diag.Ok AND NOT xIsDriveVirtualException THEN
		stIsDriveVirtualException.etDiag 	:= etDiag;
		stIsDriveVirtualException.udiDiagExt:= etDiagExt;
		stIsDriveVirtualException.sDiagExt 	:= FC_EtDiagExtToString(etDiagExt);															
		stIsDriveVirtualException.sMsg 		:= sMsgBuffer;
		xIsDriveVirtualException 			:= TRUE;
	END_IF
	
	fbExceptionHandler.SetException(i_xExceptionActive	:= xIsDriveVirtualException, 
									iq_stException		:= stIsDriveVirtualException, 
									iq_stExceptionList	:= iq_stExceptionList);
					
	xInitSuccessful := xInitSuccessful AND NOT xIsDriveVirtualException;
	etDiag := GD.ET_Diag.Ok;
//
//--- Set DeadTime compensation parameters depending on used type of Master---------------------------------------------------------
	FC_SetDeadTimeCompensation(i_stSubModuleInterfaceMain := stSlave2Interface.stMain);
	
//
//--- Set Velocity Parameters ---------------------------------------------------------
	stSlave2Interface.stMain.i_lrMotionActiveVelLimit						:= 15.0;	//--- Limit for max. velocity of astAxisModuleInterface to switch output AxisMove in Units/s ---------------------------------------------------------
	stSlave2Interface.stMain.i_etMotionActiveVelType						:= AXM.ET_MotionActiveVelType.Velocity;
	
	stSlave2Interface.stMain.stReducedVelocity.i_xEnableReducedVelocity		:= FALSE;
	stSlave2Interface.stMain.stReducedVelocity.i_xOnlyLimitCheck			:= FALSE;
	stSlave2Interface.stMain.stReducedVelocity.i_lrMaxReducedVelocity		:= 50.0;

//
//--- Stop Parameters ---------------------------------------------------------
	stSlave2Interface.stMain.i_timMasterStop								:= T#1S;
	stSlave2Interface.stMain.i_xHwLimitPos									:= FALSE;
	stSlave2Interface.stMain.i_xHwLimitNeg									:= FALSE;
	stSlave2Interface.stMain.i_xStart										:= FALSE;
//
//--- Set Homing Mode ---------------------------------------------------------
	//
	IF xDriveIsVirtual THEN
		stSlave2Interface.stHome.i_etMode := PDL.ET_HomeMode.SetPosAxisAndLogEncoderPosition;			//--- Homing Mode  in case of virtual axis ---------------------------------------------------------
	ELSE
		stSlave2Interface.stHome.i_etMode := PDL.ET_HomeMode.PosDirectionPosEdgeTp;						//--- Homing Mode in case of real axis ---------------------------------------------------------
	END_IF
		
	
	stSlave2Interface.stHome.i_xEnableInitAbsReadPos := FALSE;		(* TRUE : Restores the AxisPosition depending on the stHome.etMode
																			  If stHome.i_etMode is equal to PDL.ET_HomeMode.RestorePosFromAxisEncoder or 
																			  to PDL.ET_HomeMode.WriteAxisEncoder, the encoder of the axis is read,
																			  or else the position will be restored from the retain area *)
																			  
	stSlave2Interface.stHome.stSetpos.iq_pstRestorePosRetain := ADR(Grp_stRestorePositionAxis2);
	
	stSlave2Interface.stHome.i_xResetHomeOk := FALSE;
//
//--- Homing mode Sensor:
	(*	PDL.ET_HomeMode.PosDirectionPosEdgeSensor
		PDL.ET_HomeMode.NegDirectionPosEdgeSensor
		PDL.ET_HomeMode.NegDirectionNegEdgeSensor
		PDL.ET_HomeMode.PosDirectionNegEdgeSensor	*)

	stSlave2Interface.stHome.stSensor.i_lrHomePosition			:= 0.0;			//--- Position at the end of homing in units ---------------------------------------------------------
	stSlave2Interface.stHome.stSensor.i_lrVel					:= 10.0;		//--- Homing ceiling velocity in units/s ---------------------------------------------------------
	stSlave2Interface.stHome.stSensor.i_lrAcc					:= 1000.0;		//--- Homing acceleration in units/s^2 ---------------------------------------------------------
	stSlave2Interface.stHome.stSensor.i_lrDec					:= 1000.0;		//--- Homing deceleration in units/s^2 ---------------------------------------------------------
	stSlave2Interface.stHome.stSensor.i_lrJerk					:= 10000.0;		//--- Homing jerk in units/s^3 ---------------------------------------------------------
	stSlave2Interface.stHome.stSensor.i_lrOffset				:= 0.0;			//--- Offset from home signal in units ---------------------------------------------------------
	stSlave2Interface.stHome.stSensor.i_lrMaxTravel				:= 720.0;		//--- Max. travel for referencing by normal input ---------------------------------------------------------
	stSlave2Interface.stHome.stSensor.i_xRotativeSystem			:= FALSE;		//--- Rotative system true or false for referencing by normal input ---------------------------------------------------------
	stSlave2Interface.stHome.stSensor.i_xSensor					:= FALSE;		//--- Input for home signal. Can be a signal from a controller input. Has to be written cyclic. ---------------------------------------------------------

//--- Homing mode LimitSwitch:
	(*	PDL.ET_HomeMode.PosDirectionPosEdgeHWLimitPos		normally open contact / Closing contact
		PDL.ET_HomeMode.NegDirectionPosEdgeHWLimitNeg		normally open contact / Closing contact
		PDL.ET_HomeMode.NegDirectionNegEdgeHWLimitNeg		normally closed contact / Opening contact  
		PDL.ET_HomeMode.PosDirectionNegEdgeHWLimitPos		normally closed contact / Opening contact *)

	stSlave2Interface.stHome.stLimitSwitch.i_lrHomePosition		:= 0.0;			//--- Position at the end of homing in units ---------------------------------------------------------
	stSlave2Interface.stHome.stLimitSwitch.i_lrVel				:= 10.0;		//--- Homing ceiling velocity in units/s ---------------------------------------------------------
	stSlave2Interface.stHome.stLimitSwitch.i_lrLowVel			:= 5.0;			//--- Homing low ceiling velocity in units/s ---------------------------------------------------------
	stSlave2Interface.stHome.stLimitSwitch.i_lrAcc				:= 1000.0;		//--- Homing acceleration in units/s^2 ---------------------------------------------------------
	stSlave2Interface.stHome.stLimitSwitch.i_lrDec				:= 1000.0;		//--- Homing deceleration in units/s^2 ---------------------------------------------------------
	stSlave2Interface.stHome.stLimitSwitch.i_lrJerk				:= 10000.0;		//--- Homing jerk in units/s^3 ---------------------------------------------------------
	stSlave2Interface.stHome.stLimitSwitch.i_lrOffset			:= 0.0;			//--- Offset from home signal in units ---------------------------------------------------------
	stSlave2Interface.stHome.stLimitSwitch.i_lrMaxTravel		:= 9999.0;		//--- Max. travel for referencing normal input as a hardware limit ---------------------------------------------------------

//--- Homing mode MoveOnPos:
	(*PDL.ET_HomeMode.MoveOnPosAbs *)

	stSlave2Interface.stHome.stMoveOnPos.i_lrTarget				:= 0.0;			//--- Position at the end of homing in units ---------------------------------------------------------
	stSlave2Interface.stHome.stMoveOnPos.i_lrVel				:= 10.0;		//--- Homing ceiling velocity in units/s ---------------------------------------------------------
	stSlave2Interface.stHome.stMoveOnPos.i_lrAcc				:= 1000.0;		//--- Homing acceleration in units/s^2 ---------------------------------------------------------
	stSlave2Interface.stHome.stMoveOnPos.i_lrDec				:= 1000.0;		//--- Homing deceleration in units/s^2 ---------------------------------------------------------
	stSlave2Interface.stHome.stMoveOnPos.i_lrJerk				:= 10000.0;		//--- Homing jerk in units/s^3 ---------------------------------------------------------
	stSlave2Interface.stHome.stMoveOnPos.i_lrPeriod				:= 0.0;			//--- Period of the axis ---------------------------------------------------------
	stSlave2Interface.stHome.stMoveOnPos.i_xRotativeSystem		:= FALSE;		//--- Rotative system true or false ---------------------------------------------------------

//--- Homing mode SetPos:
	(*	PDL.ET_HomeMode.SetPosAxisPosition 
		PDL.ET_HomeMode.SetPosLogEncoderPosition 
		PDL.ET_HomeMode.SetPosAxisAndLogEncoderPosition
		PDL.ET_HomeMode.RestorePosFromAxisEncoder 
		PDL.ET_HomeMode.RestorePosFromRetain 				*)

	stSlave2Interface.stHome.stSetpos.i_lrHomePosition			:= 0.0;			//--- Position at the end of homing in units ---------------------------------------------------------
	stSlave2Interface.stHome.stSetpos.i_lrEncoderPosition		:= 0.0;			//--- Encoder position in units after homing ---------------------------------------------------------
	stSlave2Interface.stHome.stSetpos.i_lrAbsEncOffset			:= 100.0;		//--- Distance to the jump of axis encoder in units  ---------------------------------------------------------
	stSlave2Interface.stHome.stSetpos.i_lrRestoreWindow			:= 180;			//--- How far can the drive be away from is correct position ---------------------------------------------------------
	stSlave2Interface.stHome.stSetpos.i_lrUserPeriod			:= 360;			//--- Period of the axis ---------------------------------------------------------

//--- Homing mode Torque:
	(*	PDL.ET_HomeMode.PosDirectionMaxTorque 
		PDL.ET_HomeMode.NegDirectionMaxTorque *)

	stSlave2Interface.stHome.stTorque.i_lrHomePosition			:= 0.0;			//--- Position at the end of homing in units ---------------------------------------------------------
	stSlave2Interface.stHome.stTorque.i_lrVel					:= 10.0;		//--- Homing ceiling velocity in units/s ---------------------------------------------------------
	stSlave2Interface.stHome.stTorque.i_lrAcc					:= 1000.0;		//--- Homing acceleration in units/s^2 ---------------------------------------------------------
	stSlave2Interface.stHome.stTorque.i_lrDec					:= 1000.0;		//--- Homing deceleration in units/s^2 ---------------------------------------------------------
	stSlave2Interface.stHome.stTorque.i_lrJerk					:= 10000.0;		//--- Homing jerk in units/s^3 ---------------------------------------------------------
	stSlave2Interface.stHome.stTorque.i_lrOffset				:= 0.0;			//--- Offset from home signal in units ---------------------------------------------------------
	stSlave2Interface.stHome.stTorque.i_lrMaxTravel				:= 9999.0;		//--- Max. travel for referencing by torque ---------------------------------------------------------
	stSlave2Interface.stHome.stTorque.i_lrMaxTorque				:= 0.0;			//--- Torque for stop in Nm / referencing by torque ---------------------------------------------------------
	stSlave2Interface.stHome.stTorque.i_diTorqueTime			:= 5;			//--- Time in msec to hold torque ---------------------------------------------------------

//--- Homing mode TouchProbe:
	(*	PDL.ET_HomeMode.PosDirectionPosEdgeTp 
		PDL.ET_HomeMode.NegDirectionPosEdgeTp 
		PDL.ET_HomeMode.NegDirectionNegEdgeTp 
		PDL.ET_HomeMode.PosDirectionNegEdgeTp *)

	stSlave2Interface.stHome.stTouchProbe.i_lrHomePosition		:= 0.0;			//--- Position at the end of homing in units ---------------------------------------------------------
	stSlave2Interface.stHome.stTouchProbe.i_lrVel				:= 100.0;		//--- Homing ceiling velocity in units/s ---------------------------------------------------------
	stSlave2Interface.stHome.stTouchProbe.i_lrAcc				:= 1000.0;		//--- Homing acceleration in units/s^2 ---------------------------------------------------------
	stSlave2Interface.stHome.stTouchProbe.i_lrDec				:= 1000.0;		//--- Homing deceleration in units/s^2 ---------------------------------------------------------
	stSlave2Interface.stHome.stTouchProbe.i_lrJerk				:= 10000.0;		//--- Homing jerk in units/s^3 ---------------------------------------------------------
	stSlave2Interface.stHome.stTouchProbe.i_lrOffset			:= 30.0;		//--- Offset from home signal in units ---------------------------------------------------------
	stSlave2Interface.stHome.stTouchProbe.i_lrMaxTravel			:= 720.0;		//--- Max. travel for referencing by TP ---------------------------------------------------------
	stSlave2Interface.stHome.stTouchProbe.i_xRotativeSystem		:= TRUE;		//--- Rotative system true or false for referencing by TP ---------------------------------------------------------
	stSlave2Interface.stHome.stTouchProbe.i_ifTouchProbe		:= TP_1;		//--- Input for TP ---------------------------------------------------------

//--- Homing mode WritePos:
	(*	PDL.ET_HomeMode.WriteAxisEncoder *)

	stSlave2Interface.stHome.stWritePos.i_lrHomePosition		:= 0.0;			//--- Position at the end of homing in units ---------------------------------------------------------
	stSlave2Interface.stHome.stWritePos.i_lrUserPeriod			:= 0.0;			//--- Calculates Drive.Position into period ( units ) ---------------------------------------------------------
	stSlave2Interface.stHome.stWritePos.i_lrAbsEncOffset		:= 100.0;		//--- Distance to the jump of axis encoder in units ---------------------------------------------------------

//
//--- Manual ---------------------------------------------------------
	//
	stSlave2Interface.stManual.i_lrVel								:= 50.0;			//--- Velocity in units/s ---------------------------------------------------------
	stSlave2Interface.stManual.i_lrAcc								:= 100.0;			//--- Acceleration in units/s^2 ---------------------------------------------------------
	stSlave2Interface.stManual.i_lrDec								:= 100.0;			//--- Deceleration in units/s^2 ---------------------------------------------------------
	stSlave2Interface.stManual.i_lrJerk								:= 1000.0;			//--- Jerk in units/s^3 ---------------------------------------------------------
	stSlave2Interface.stManual.i_lrMaxDistance						:= 120.0;			//--- Max pathlengths for one step in units ---------------------------------------------------------
	stSlave2Interface.stManual.i_xEndless							:= FALSE;			//--- TRUE: jogging endless; Position between the periode; FALSE: jogging in steps. Position can be out of periode ---------------------------------------------------------
	stSlave2Interface.stManual.i_lrPeriod							:= 360.0;			//--- Period of the axis ---------------------------------------------------------

//
//--- Cam ---------------------------------------------------------
	//
	stSlave2Interface.stMultiCam.i_etCSModeSlave					:= PDL.ET_MultiCamCsModeSlave.SetSlavePositionToFirstCamPosition;		//--- ColdStartMode Slave ---------------------------------------------------------
	stSlave2Interface.stMultiCam.i_etCSModeMaster					:= PDL.ET_MultiCamCsModeMaster.SetMasterPositionToFirstCamPosition;		//--- ColdStartMode Master ---------------------------------------------------------
	stSlave2Interface.stMultiCam.i_etWSMode							:= PDL.ET_MultiCamWsMode.StoredCamMoveAlwaysNoPositionCheck;			//--- WarmStartMode ---------------------------------------------------------
	stSlave2Interface.stMultiCam.i_lrWSWindow						:= 5.0;											//--- WarmStartWindow in Axis units ---------------------------------------------------------
	stSlave2Interface.stMultiCam.i_lrWSVel							:= 100.0;										//--- Velocity for WarmStart and CSModeSlave = PDL.ET_MultiCamCsModeSlave.MoveSlaveToFirstCamPosition in Units/s ---------------------------------------------------------
	stSlave2Interface.stMultiCam.i_lrWSAcc							:= 1000.0;										//--- Acceleration and deceleration for Warmstart and CSModeSlave = PDL.ET_MultiCamCsModeSlave.MoveSlaveToFirstCamPosition in Units/s^2 ---------------------------------------------------------
	stSlave2Interface.stMultiCam.i_lrWSJerk							:= 10000.0;										//--- Jerk for Warmstart and CSModeSlave = PDL.ET_MultiCamCsModeSlave.MoveSlaveToFirstCamPosition in units/s^3 ---------------------------------------------------------
	stSlave2Interface.stMultiCam.i_diTXend							:= 2*SYSTEMINTERFACE.FC_LzsTaskGetInterval();	//--- Time of XLowEnd and XHighEnd befor Xend or Xstart in msec---------------------------------------------------------
	stSlave2Interface.stMultiCam.i_lrInstantXLimMax					:= 0.0;											//--- Switch off position at 'InstantNewCam' ---------------------------------------------------------
	
	stSlave2Interface.stMultiCam.i_xEnableTabHandler				:= TRUE;										//--- TRUE: TabHandler is enabled ---------------------------------------------------------
	stSlave2Interface.stMultiCam.i_udiTableSelectNr					:= AXM.ET_ParId.User;							//--- Number of table which is used in the next cycle ---------------------------------------------------------
	
	stSlave2Interface.stMultiCam.i_xSetEncoderParameters			:= FALSE;										//--- TRUE: The parameters MasterId, FeedConstand, GearIn and GearOut will be copyed into LEnc object ---------------------------------------------------------
	stSlave2Interface.stMultiCam.i_xSetEncoderPosition				:= TRUE;										//--- TRUE: Manipulation of LEnc object on startup OpMode MultiCam ---------------------------------------------------------
	stSlave2Interface.stMultiCam.i_lrSetEncoderOffset				:= 0.0;											//--- Master encoder offset ---------------------------------------------------------
	stSlave2Interface.stMultiCam.i_xCheckEncoderPeriod				:= TRUE;										//--- TRUE: Check of encoder period = 0. If encoder period <> 0 -> Exception ---------------------------------------------------------
	
	//--- stSlave2Interface.stMultiCam.iq_xNewCam						:= FALSE;									//--- TRUE: A new DataStruct will be load for next cycle. Will be reset when new cycle is started in case of stMultiCam.i_xEnableTabHandler = FALSE. ---------------------------------------------------------
	//--- stSlave2Interface.stMultiCam.iq_xInstantNewCam				:= FALSE;									//--- TRUE: A new DataStruct will be load. It will be active at master position stMultiCam.i_lrInstantXLimMax. Will be reset when ne DataStruct is active ---------------------------------------------------------
	//--- stSlave2Interface.stMultiCam.iq_xChangeMaster				:= FALSE;										//--- TRUE: Switch to a new Master. Will be reset when done. ---------------------------------------------------------			
	
	//--- stSlave2Interface.stMultiCam.iq_stExt		;						//--- Extended In of the Multicam FB, can be used if needed! ---------------------------------------------------------
	
	//--- DataStruct used in CamDiagram_Slave2 ---------------------------------------------------------
	//stSlave2Interface.stMultiCam.iq_astMotionPar[AXM.ET_ParId.User].diNumberOfCamPoints		:= 4;	
	//stSlave2Interface.stMultiCam.iq_astMotionPar[AXM.ET_ParId.User].lrYPeriod				:= 0.0;
	//
	//stSlave2Interface.stMultiCam.iq_astMotionPar[AXM.ET_ParId.User].astCamPoint[0].lrX		:= 0.0;
	//stSlave2Interface.stMultiCam.iq_astMotionPar[AXM.ET_ParId.User].astCamPoint[0].lrY		:= 0.0;
	//stSlave2Interface.stMultiCam.iq_astMotionPar[AXM.ET_ParId.User].astCamPoint[0].lrM		:= 0.0;
	//stSlave2Interface.stMultiCam.iq_astMotionPar[AXM.ET_ParId.User].astCamPoint[0].etCamType	:= PDL.ET_CamType.Poly5Com;
	//stSlave2Interface.stMultiCam.iq_astMotionPar[AXM.ET_ParId.User].astCamPoint[1].lrX		:= 60.0;
	//stSlave2Interface.stMultiCam.iq_astMotionPar[AXM.ET_ParId.User].astCamPoint[1].lrY		:= 30.0;
	//stSlave2Interface.stMultiCam.iq_astMotionPar[AXM.ET_ParId.User].astCamPoint[1].lrM		:= 1.0;
	//stSlave2Interface.stMultiCam.iq_astMotionPar[AXM.ET_ParId.User].astCamPoint[1].etCamType	:= PDL.ET_CamType.Straight;
	//stSlave2Interface.stMultiCam.iq_astMotionPar[AXM.ET_ParId.User].astCamPoint[2].lrX		:= 240.0;
	//stSlave2Interface.stMultiCam.iq_astMotionPar[AXM.ET_ParId.User].astCamPoint[2].lrY		:= 210.0;
	//stSlave2Interface.stMultiCam.iq_astMotionPar[AXM.ET_ParId.User].astCamPoint[2].lrM		:= 1.0;
	//stSlave2Interface.stMultiCam.iq_astMotionPar[AXM.ET_ParId.User].astCamPoint[2].etCamType	:= PDL.ET_CamType.Poly5Com;
	//stSlave2Interface.stMultiCam.iq_astMotionPar[AXM.ET_ParId.User].astCamPoint[3].lrX		:= 360.0;
	//stSlave2Interface.stMultiCam.iq_astMotionPar[AXM.ET_ParId.User].astCamPoint[3].lrY		:= 0.0;
	//stSlave2Interface.stMultiCam.iq_astMotionPar[AXM.ET_ParId.User].astCamPoint[3].lrM		:= 0.0;
	//stSlave2Interface.stMultiCam.iq_astMotionPar[AXM.ET_ParId.User].astCamPoint[3].etCamType	:= PDL.ET_CamType.Poly5Com;
	
	stSlave2Interface.stMultiCam.iq_astMotionPar[AXM.ET_ParId.Idle].diUserTableId	:= UDINT_TO_DINT(AXM.ET_ParId.Idle);
	stSlave2Interface.stMultiCam.iq_astMotionPar[AXM.ET_ParId.Start].diUserTableId	:= UDINT_TO_DINT(AXM.ET_ParId.Start);
	stSlave2Interface.stMultiCam.iq_astMotionPar[AXM.ET_ParId.Cont].diUserTableId	:= UDINT_TO_DINT(AXM.ET_ParId.Cont);
	stSlave2Interface.stMultiCam.iq_astMotionPar[AXM.ET_ParId.Stop].diUserTableId	:= UDINT_TO_DINT(AXM.ET_ParId.Stop);
	stSlave2Interface.stMultiCam.iq_astMotionPar[AXM.ET_ParId.User].diUserTableId	:= UDINT_TO_DINT(AXM.ET_ParId.User);


	//--- ILS Data --------------------------------------------------------
	//---
	//stSlave2Interface.stMultiCam.i_udiIlsSlaveNumber													:= 1;
	//
	//G_stIlsData.i_stRunTime.astSlaveLimits[stSlave2Interface.stMultiCam.i_udiIlsSlaveNumber].lrPosVel	:= 1000.0;
	//G_stIlsData.i_stRunTime.astSlaveLimits[stSlave2Interface.stMultiCam.i_udiIlsSlaveNumber].lrNegVel	:= -1000.0;
	//G_stIlsData.i_stRunTime.astSlaveLimits[stSlave2Interface.stMultiCam.i_udiIlsSlaveNumber].lrPosAcc	:= 10000.0;
	//G_stIlsData.i_stRunTime.astSlaveLimits[stSlave2Interface.stMultiCam.i_udiIlsSlaveNumber].lrNegAcc	:= -10000.0;
	//
	//G_stIlsData.i_astCamData[stSlave2Interface.stMultiCam.i_udiIlsSlaveNumber].diNumberOfMasterPeriods	:= 1;	
	//G_stIlsData.i_astCamData[stSlave2Interface.stMultiCam.i_udiIlsSlaveNumber].diMasterPeriodInit		:= 1;
	//G_stIlsData.i_astCamData[stSlave2Interface.stMultiCam.i_udiIlsSlaveNumber].lrXOffset				:= 0.0;
	//
	//stSlave2Interface.stMultiCam.pstIlsData																:= ADR(G_stIlsData);
//
//--- Endless ---------------------------------------------------------
	//
	stSlave2Interface.stEndless.i_lrVel								:= 100.0;			//--- Velocity in Units/s ---------------------------------------------------------
	stSlave2Interface.stEndless.i_lrAcc								:= 1000.0;			//--- Acceleration in Units/s^2 ---------------------------------------------------------
	stSlave2Interface.stEndless.i_lrDec								:= 1000.0;			//--- Deceleration in Units/s^2 ---------------------------------------------------------
	stSlave2Interface.stEndless.i_lrJerk							:= 10000.0;			//--- Jerk in units/s^3 ---------------------------------------------------------
	stSlave2Interface.stEndless.i_lrPeriod							:= 360.0;			//--- Period one cycle in units ---------------------------------------------------------
	stSlave2Interface.stEndless.i_lrStopPosition					:= 0.5;				//--- Stop position in units ---------------------------------------------------------
//
//--- Endless ILS ---------------------------------------------------------
	//
	//G_stIlsData.i_stConfig.diNumberOfSlaves							:= 0;
	//G_stIlsData.i_stConfig.diPositionGridSize						:= 500;
	//G_stIlsData.i_stConfig.diTimeGridSize							:= 50;
	//G_stIlsData.i_stConfig.lrHysteresis								:= 20;
	//
	//G_stIlsData.i_stRunTime.iMasterAverageVelocityCycles			:= 10;
	//G_stIlsData.i_stRunTime.lrMasterMaxAbsVel						:= 100.0;
	//G_stIlsData.i_stRunTime.lrMasterMaxAbsAcc						:= 1000.0;
	//G_stIlsData.i_stRunTime.lrMasterMaxAbsJerk						:= 10000.0;
	//G_stIlsData.i_stRunTime.xActivateLimitation						:= TRUE;
	//
	//stSlave2Interface.stEndless.pstIlsData							:= ADR(G_stIlsData);
//
//--- Pos ---------------------------------------------------------
	//
	stSlave2Interface.stPos.i_etPosMode								:= SYSTEMINTERFACE.ET_PosMode.Relative;			//--- SYSTEMINTERFACE.ET_PosMode.Endless, SYSTEMINTERFACE.ET_PosMode.Relative, SYSTEMINTERFACE.ET_PosMode.Absolute ---------------------------------------------------------
	stSlave2Interface.stPos.i_lrTarget								:= -360.0;										//--- Target position or distance in Units ---------------------------------------------------------
	stSlave2Interface.stPos.i_lrVel									:= 100.0;										//--- Ceiling velocity in Units/s ---------------------------------------------------------
	stSlave2Interface.stPos.i_lrAcc									:= 3600.0;										//--- Acceleration in Units/s^2 ---------------------------------------------------------
	stSlave2Interface.stPos.i_lrDec									:= 3600.0;										//--- Deceleration in Units/s^2 ---------------------------------------------------------
	stSlave2Interface.stPos.i_lrJerk								:= 36000.0;										//--- Jerk in units/s^3 ---------------------------------------------------------

	//--- stSlave2Interface.stPos.i_xStop								:= FALSE;
//
//--- End of system generated code, could be modified for your application ---------------------------------------------------------
END_ACTION

ACTION Init_CmdTables:
//- System generated code, could be modified FOR your application -

//-------------------------------------------------------------------------------------------------------------------
//-- Prepare  --
	//
	TPL.FC_FirstStep(udiStepIndex, diStep);
	astPrepareTable[udiStepIndex].sTitle					:= 'DriveEnable On AllSubModules';
	astPrepareTable[udiStepIndex].udiModuleName				:= TPL.Gc_udiAllSubModules;
	astPrepareTable[udiStepIndex].diStep					:= diStep;
	astPrepareTable[udiStepIndex].diCMD						:= AXM.ET_Cmd.DriveEnableOn;
	astPrepareTable[udiStepIndex].timTimeOut				:= T#0MS;
	astPrepareTable[udiStepIndex].xEndCMD					:= FALSE;
	
	TPL.FC_NextStep(udiStepIndex, diStep);
	astPrepareTable[udiStepIndex].sTitle					:= 'Homing Mode AllSubModules';
	astPrepareTable[udiStepIndex].udiModuleName				:= TPL.Gc_udiAllSubModules;
	astPrepareTable[udiStepIndex].diStep					:= diStep;
	astPrepareTable[udiStepIndex].diCMD						:= AXM.ET_Cmd.Homing;
	astPrepareTable[udiStepIndex].timTimeOut				:= T#0MS;
	astPrepareTable[udiStepIndex].xEndCMD					:= FALSE;
	
	TPL.FC_NextStep(udiStepIndex, diStep);
	astPrepareTable[udiStepIndex].sTitle					:= 'Homing Start AllSubModules';
	astPrepareTable[udiStepIndex].udiModuleName				:= TPL.Gc_udiAllSubModules;
	astPrepareTable[udiStepIndex].diStep					:= diStep;
	astPrepareTable[udiStepIndex].diCMD						:= AXM.ET_Cmd.Start;
	astPrepareTable[udiStepIndex].timTimeOut				:= T#0MS;
	astPrepareTable[udiStepIndex].xEndCMD					:= FALSE;
	
	TPL.FC_LastStep(udiStepIndex, diStep);
	astPrepareTable[udiStepIndex].sTitle					:= 'End';
	astPrepareTable[udiStepIndex].udiModuleName				:= 0;
	astPrepareTable[udiStepIndex].diStep					:= diStep;
	astPrepareTable[udiStepIndex].diCMD						:= 0;
	astPrepareTable[udiStepIndex].timTimeOut				:= T#0MS;
	astPrepareTable[udiStepIndex].xEndCMD					:= TRUE;
	
	TPL.FC_FirstCmdTable(iq_udiTableIndex:= udiTableIndex);
	astListofCMDTables[udiTableIndex].sTitle				:= 'Prepare';
	astListofCMDTables[udiTableIndex].diCMD					:= ET_Cmd.Prepare;
	astListofCMDTables[udiTableIndex].udiNumberOfCmdSteps	:= udiStepIndex;

//-------------------------------------------------------------------------------------------------------------------
//-- Auto  --
	//
	TPL.FC_FirstStep(udiStepIndex, diStep);
	astAutoTable[udiStepIndex].sTitle						:= 'DriveEnable On AllSubModules';
	astAutoTable[udiStepIndex].udiModuleName				:= TPL.Gc_udiAllSubModules;
	astAutoTable[udiStepIndex].diStep						:= diStep;
	astAutoTable[udiStepIndex].diCMD						:= AXM.ET_Cmd.DriveEnableOn;
	astAutoTable[udiStepIndex].timTimeOut					:= T#0MS;
	astAutoTable[udiStepIndex].xEndCMD						:= FALSE;
	
	TPL.FC_NextStep(udiStepIndex, diStep);
	astAutoTable[udiStepIndex].sTitle						:= 'Cam WS Mode AllSubModules';
	astAutoTable[udiStepIndex].udiModuleName				:= TPL.Gc_udiAllSubModules;
	astAutoTable[udiStepIndex].diStep						:= diStep;
	astAutoTable[udiStepIndex].diCMD						:= AXM.ET_Cmd.CamWs;
	astAutoTable[udiStepIndex].timTimeOut					:= T#0MS;
	astAutoTable[udiStepIndex].xEndCMD						:= FALSE;
	
	TPL.FC_NextStep(udiStepIndex, diStep);
	astAutoTable[udiStepIndex].sTitle						:= 'Start AllSubModules';
	astAutoTable[udiStepIndex].udiModuleName				:= TPL.Gc_udiAllSubModules;
	astAutoTable[udiStepIndex].diStep						:= diStep;
	astAutoTable[udiStepIndex].diCMD						:= AXM.ET_Cmd.Start;
	astAutoTable[udiStepIndex].timTimeOut					:= T#0MS;
	astAutoTable[udiStepIndex].xEndCMD						:= FALSE;
	
	TPL.FC_NextStep(udiStepIndex, diStep);
	astAutoTable[udiStepIndex].sTitle						:= 'WarmStart AllSubModules';
	astAutoTable[udiStepIndex].udiModuleName				:= TPL.Gc_udiAllSubModules;
	astAutoTable[udiStepIndex].diStep						:= diStep;
	astAutoTable[udiStepIndex].diCMD						:= AXM.ET_Cmd.WsStart;
	astAutoTable[udiStepIndex].timTimeOut					:= T#0MS;
	astAutoTable[udiStepIndex].xEndCMD						:= FALSE;
	
	TPL.FC_LastStep(udiStepIndex, diStep);
	astAutoTable[udiStepIndex].sTitle						:= 'End';
	astAutoTable[udiStepIndex].udiModuleName				:= 0;
	astAutoTable[udiStepIndex].diStep						:= diStep;
	astAutoTable[udiStepIndex].diCMD						:= 0;
	astAutoTable[udiStepIndex].timTimeOut					:= T#0MS;
	astAutoTable[udiStepIndex].xEndCMD						:= TRUE;
	
	TPL.FC_NextCmdTable(iq_udiTableIndex:= udiTableIndex);
	astListofCMDTables[udiTableIndex].sTitle				:= 'Auto';
	astListofCMDTables[udiTableIndex].diCMD					:= ET_Cmd.Auto;
	astListofCMDTables[udiTableIndex].udiNumberOfCmdSteps	:= udiStepIndex;

//-------------------------------------------------------------------------------------------------------------------
//-- Manual  --
	//
	TPL.FC_FirstStep(udiStepIndex, diStep);
	astManualTable[udiStepIndex].sTitle						:= 'DriveEnable On AllSubModules';
	astManualTable[udiStepIndex].udiModuleName				:= TPL.Gc_udiAllSubModules;
	astManualTable[udiStepIndex].diStep						:= diStep;
	astManualTable[udiStepIndex].diCMD						:= AXM.ET_Cmd.DriveEnableOn;
	astManualTable[udiStepIndex].timTimeOut					:= T#0MS;
	astManualTable[udiStepIndex].xEndCMD					:= FALSE;
	
	TPL.FC_NextStep(udiStepIndex, diStep);
	astManualTable[udiStepIndex].sTitle						:= 'Manual Mode AllSubModules';
	astManualTable[udiStepIndex].udiModuleName				:= TPL.Gc_udiAllSubModules;
	astManualTable[udiStepIndex].diStep						:= diStep;
	astManualTable[udiStepIndex].diCMD						:= AXM.ET_Cmd.Manual;
	astManualTable[udiStepIndex].timTimeOut					:= T#0MS;
	astManualTable[udiStepIndex].xEndCMD					:= FALSE;
	
	TPL.FC_LastStep(udiStepIndex, diStep);
	astManualTable[udiStepIndex].sTitle						:= 'End';
	astManualTable[udiStepIndex].udiModuleName				:= 0;
	astManualTable[udiStepIndex].diStep						:= diStep;
	astManualTable[udiStepIndex].diCMD						:= 0;
	astManualTable[udiStepIndex].timTimeOut					:= T#0MS;
	astManualTable[udiStepIndex].xEndCMD					:= TRUE;
	
	TPL.FC_NextCmdTable(iq_udiTableIndex:= udiTableIndex);
	astListofCMDTables[udiTableIndex].sTitle				:= 'Manual';
	astListofCMDTables[udiTableIndex].diCMD					:= ET_Cmd.Manual;
	astListofCMDTables[udiTableIndex].udiNumberOfCmdSteps	:= udiStepIndex;

